LIN {X 0,Y 390.142,Z 309.368,A -85,B 0,C 180,E1 -11537.308,E2 -11537.308} C_VEL
LIN {X 0,Y 390.081,Z 309.382,A -85,B 0,C 180,E1 -11540.471,E2 -11540.471} C_VEL
LIN {X 0,Y 390.069,Z 309.39,A -85,B 0,C 180,E1 -11544.482,E2 -11544.482} C_VEL
LIN {X 0,Y 390.112,Z 309.375,A -85,B 0,C 180,E1 -11547.931,E2 -11547.931} C_VEL
LIN {X 0,Y 390.017,Z 309.4,A -85,B 0,C 180,E1 -11551.506,E2 -11551.506} C_VEL
LIN {X 0,Y 390.065,Z 309.388,A -85,B 0,C 180,E1 -11555.21,E2 -11555.21} C_VEL
LIN {X 0,Y 390.082,Z 309.386,A -85,B 0,C 180,E1 -11559.094,E2 -11559.094} C_VEL
LIN {X 0,Y 390.039,Z 309.401,A -85,B 0,C 180,E1 -11562.375,E2 -11562.375} C_VEL
LIN {X 0,Y 390.041,Z 309.396,A -85,B 0,C 180,E1 -11565.355,E2 -11565.355} C_VEL
LIN {X 0,Y 390.021,Z 309.39,A -85,B 0,C 180,E1 -11568.187,E2 -11568.187} C_VEL
LIN {X 0,Y 390.061,Z 309.392,A -85,B 0,C 180,E1 -11570.905,E2 -11570.905} C_VEL
LIN {X 0,Y 390.084,Z 309.385,A -85,B 0,C 180,E1 -11574.794,E2 -11574.794} C_VEL
LIN {X 0,Y 390.028,Z 309.401,A -85,B 0,C 180,E1 -11578.497,E2 -11578.497} C_VEL
LIN {X 0,Y 390.13,Z 309.588,A -85,B 0,C 180,E1 -11579.709,E2 -11579.709} C_VEL
LIN {X 0,Y 392.282,Z 320.516,A -85,B 0,C 180,E1 -11583.105,E2 -11583.105} C_VEL
LIN {X 0,Y 392.85,Z 325.729,A -85,B 0,C 180,E1 -11584.574,E2 -11584.574} C_VEL
LIN {X 0,Y 391.795,Z 337.996,A -85,B 0,C 180,E1 -11587.871,E2 -11587.871} C_VEL
LIN {X 0,Y 391.304,Z 343.848,A -85,B 0,C 180,E1 -11589.465,E2 -11589.465} C_VEL
LIN {X 0,Y 391.869,Z 347.073,A -85,B 0,C 180,E1 -11589.616,E2 -11589.616} C_VEL
LIN {X 0,Y 396.698,Z 373.255,A -85,B 0,C 180,E1 -11590.366,E2 -11590.366} C_VEL
LIN {X 0,Y 396.546,Z 399.29,A -85,B 0,C 180,E1 -11590.847,E2 -11590.847} C_VEL
LIN {X 0,Y 395.821,Z 450.139,A -85,B 0,C 180,E1 -11591.797,E2 -11591.797} C_VEL
LIN {X 0,Y 395.391,Z 460.446,A -85,B 0,C 180,E1 -11592.112,E2 -11592.112} C_VEL
LIN {X 0,Y 394.883,Z 469.958,A -85,B 0,C 180,E1 -11592.523,E2 -11592.523} C_VEL
LIN {X 0,Y 394.257,Z 480.039,A -85,B 0,C 180,E1 -11593.095,E2 -11593.095} C_VEL
LIN {X 0,Y 393.494,Z 489.796,A -85,B 0,C 180,E1 -11593.796,E2 -11593.796} C_VEL
LIN {X 0,Y 392.668,Z 499.864,A -85,B 0,C 180,E1 -11594.693,E2 -11594.693} C_VEL
LIN {X 0,Y 391.74,Z 510.864,A -85,B 0,C 180,E1 -11595.915,E2 -11595.915} C_VEL
LIN {X 0,Y 390.927,Z 520.506,A -85,B 0,C 180,E1 -11597.278,E2 -11597.278} C_VEL
LIN {X 0,Y 390.31,Z 526.707,A -85,B 0,C 180,E1 -11598.313,E2 -11598.313} C_VEL
LIN {X 0,Y 389.792,Z 533.245,A -85,B 0,C 180,E1 -11599.613,E2 -11599.613} C_VEL
LIN {X 0,Y 389.389,Z 537.746,A -85,B 0,C 180,E1 -11600.652,E2 -11600.652} C_VEL
LIN {X 0,Y 389.034,Z 543.238,A -85,B 0,C 180,E1 -11602.213,E2 -11602.213} C_VEL
LIN {X 0,Y 388.796,Z 547.562,A -85,B 0,C 180,E1 -11603.774,E2 -11603.774} C_VEL
LIN {X 0,Y 388.741,Z 549.929,A -85,B 0,C 180,E1 -11604.814,E2 -11604.814} C_VEL
LIN {X 0,Y 388.701,Z 551.728,A -85,B 0,C 180,E1 -11605.853,E2 -11605.853} C_VEL
LIN {X 0,Y 388.661,Z 554.171,A -85,B 0,C 180,E1 -11607.927,E2 -11607.927} C_VEL
LIN {X 0,Y 388.704,Z 554.761,A -85,B 0,C 180,E1 -11608.964,E2 -11608.964} C_VEL
LIN {X 0,Y 388.704,Z 554.761,A -85,B 0,C 180,E1 -11611.036,E2 -11611.036} C_VEL
LIN {X 0,Y 388.661,Z 554.171,A -85,B 0,C 180,E1 -11612.073,E2 -11612.073} C_VEL
LIN {X 0,Y 388.701,Z 551.728,A -85,B 0,C 180,E1 -11614.147,E2 -11614.147} C_VEL
LIN {X 0,Y 388.727,Z 548.672,A -85,B 0,C 180,E1 -11615.752,E2 -11615.752} C_VEL
LIN {X 0,Y 388.94,Z 544.792,A -85,B 0,C 180,E1 -11617.266,E2 -11617.266} C_VEL
LIN {X 0,Y 389.257,Z 539.662,A -85,B 0,C 180,E1 -11618.828,E2 -11618.828} C_VEL
LIN {X 0,Y 389.666,Z 534.4,A -85,B 0,C 180,E1 -11620.128,E2 -11620.128} C_VEL
LIN {X 0,Y 390.165,Z 528.082,A -85,B 0,C 180,E1 -11621.428,E2 -11621.428} C_VEL
LIN {X 0,Y 390.767,Z 522.133,A -85,B 0,C 180,E1 -11622.463,E2 -11622.463} C_VEL
LIN {X 0,Y 391.353,Z 515.204,A -85,B 0,C 180,E1 -11623.5,E2 -11623.5} C_VEL
LIN {X 0,Y 392.026,Z 507.023,A -85,B 0,C 180,E1 -11624.535,E2 -11624.535} C_VEL
LIN {X 0,Y 392.753,Z 498.511,A -85,B 0,C 180,E1 -11625.436,E2 -11625.436} C_VEL
LIN {X 0,Y 393.496,Z 489.796,A -85,B 0,C 180,E1 -11626.204,E2 -11626.204} C_VEL
LIN {X 0,Y 394.264,Z 480.04,A -85,B 0,C 180,E1 -11626.904,E2 -11626.904} C_VEL
LIN {X 0,Y 394.855,Z 469.958,A -85,B 0,C 180,E1 -11627.479,E2 -11627.479} C_VEL
LIN {X 0,Y 395.422,Z 460.447,A -85,B 0,C 180,E1 -11627.887,E2 -11627.887} C_VEL
LIN {X 0,Y 395.803,Z 450.139,A -85,B 0,C 180,E1 -11628.203,E2 -11628.203} C_VEL
LIN {X 0,Y 396.422,Z 404.772,A -85,B 0,C 180,E1 -11629.056,E2 -11629.056} C_VEL
LIN {X 0,Y 396.829,Z 373.982,A -85,B 0,C 180,E1 -11629.614,E2 -11629.614} C_VEL
LIN {X 0,Y 391.498,Z 345.223,A -85,B 0,C 180,E1 -11630.439,E2 -11630.439} C_VEL
LIN {X 0,Y 391.324,Z 343.641,A -85,B 0,C 180,E1 -11630.568,E2 -11630.568} C_VEL
LIN {X 0,Y 392.44,Z 331.107,A -85,B 0,C 180,E1 -11634.029,E2 -11634.029} C_VEL
LIN {X 0,Y 392.897,Z 325.998,A -85,B 0,C 180,E1 -11635.423,E2 -11635.423} C_VEL
LIN {X 0,Y 392.326,Z 320.813,A -85,B 0,C 180,E1 -11636.892,E2 -11636.892} C_VEL
LIN {X 0,Y 390.56,Z 311.768,A -85,B 0,C 180,E1 -11639.599,E2 -11639.599} C_VEL
LIN {X 0,Y 390.097,Z 309.445,A -85,B 0,C 180,E1 -11640.369,E2 -11640.369} C_VEL
LIN {X 0,Y 390.068,Z 309.4,A -85,B 0,C 180,E1 -11644.024,E2 -11644.024} C_VEL
LIN {X 0,Y 390.039,Z 309.399,A -85,B 0,C 180,E1 -11647.549,E2 -11647.549} C_VEL
LIN {X 0,Y 390.02,Z 309.382,A -85,B 0,C 180,E1 -11650.814,E2 -11650.814} C_VEL
LIN {X 0,Y 390.051,Z 309.401,A -85,B 0,C 180,E1 -11653.885,E2 -11653.885} C_VEL
LIN {X 0,Y 390.054,Z 309.395,A -85,B 0,C 180,E1 -11656.789,E2 -11656.789} C_VEL
LIN {X 0,Y 390.053,Z 309.392,A -85,B 0,C 180,E1 -11659.559,E2 -11659.559} C_VEL
LIN {X 0,Y 390.038,Z 309.398,A -85,B 0,C 180,E1 -11662.449,E2 -11662.449} C_VEL
LIN {X 0,Y 390.056,Z 309.384,A -85,B 0,C 180,E1 -11666.043,E2 -11666.043} C_VEL
LIN {X 0,Y 390.041,Z 309.399,A -85,B 0,C 180,E1 -11669.868,E2 -11669.868} C_VEL
LIN {X 0,Y 390.107,Z 309.372,A -85,B 0,C 180,E1 -11673.231,E2 -11673.231} C_VEL
LIN {X 0,Y 390.061,Z 309.393,A -85,B 0,C 180,E1 -11676.763,E2 -11676.763} C_VEL
LIN {X 0,Y 390.097,Z 309.375,A -85,B 0,C 180,E1 -11679.982,E2 -11679.982} C_VEL
LIN {X 0,Y 390.131,Z 309.374,A -85,B 0,C 180,E1 -11683.247,E2 -11683.247} C_VEL
LIN {X 0,Y 390.187,Z 309.377,A -85,B 0,C 180,E1 -11686.561,E2 -11686.561} C_VEL
LIN {X 0,Y 390.197,Z 309.351,A -85,B 0,C 180,E1 -11690.67,E2 -11690.67} C_VEL
LIN {X 0,Y 390.318,Z 309.363,A -85,B 0,C 180,E1 -11693.797,E2 -11693.797} C_VEL
LIN {X 0,Y 390.412,Z 309.342,A -85,B 0,C 180,E1 -11697.936,E2 -11697.936} C_VEL
LIN {X 0,Y 390.54,Z 309.307,A -85,B 0,C 180,E1 -11699.999,E2 -11699.999} C_VEL
LIN {X 0,Y 390.302,Z 309.359,A -85,B 0,C 180,E1 -11703.096,E2 -11703.096} C_VEL
LIN {X 0,Y 390.292,Z 309.361,A -85,B 0,C 180,E1 -11706.66,E2 -11706.66} C_VEL
LIN {X 0,Y 390.196,Z 309.354,A -85,B 0,C 180,E1 -11709.328,E2 -11709.328} C_VEL
LIN {X 0,Y 390.185,Z 309.381,A -85,B 0,C 180,E1 -11713.438,E2 -11713.438} C_VEL
LIN {X 0,Y 390.139,Z 309.375,A -85,B 0,C 180,E1 -11717.307,E2 -11717.307} C_VEL
LIN {X 0,Y 390.079,Z 309.378,A -85,B 0,C 180,E1 -11720.47,E2 -11720.47} C_VEL
LIN {X 0,Y 390.08,Z 309.394,A -85,B 0,C 180,E1 -11723.351,E2 -11723.351} C_VEL
LIN {X 0,Y 390.104,Z 309.376,A -85,B 0,C 180,E1 -11726.768,E2 -11726.768} C_VEL
LIN {X 0,Y 390.035,Z 309.398,A -85,B 0,C 180,E1 -11730.299,E2 -11730.299} C_VEL
LIN {X 0,Y 390.059,Z 309.386,A -85,B 0,C 180,E1 -11734.025,E2 -11734.025} C_VEL
LIN {X 0,Y 390.039,Z 309.399,A -85,B 0,C 180,E1 -11737.552,E2 -11737.552} C_VEL
LIN {X 0,Y 390.074,Z 309.386,A -85,B 0,C 180,E1 -11740.826,E2 -11740.826} C_VEL
LIN {X 0,Y 390.094,Z 309.391,A -85,B 0,C 180,E1 -11743.894,E2 -11743.894} C_VEL
LIN {X 0,Y 390.049,Z 309.362,A -85,B 0,C 180,E1 -11747.624,E2 -11747.624} C_VEL
LIN {X 0,Y 390.087,Z 309.392,A -85,B 0,C 180,E1 -11750.908,E2 -11750.908} C_VEL
LIN {X 0,Y 390.079,Z 309.371,A -85,B 0,C 180,E1 -11754.793,E2 -11754.793} C_VEL
LIN {X 0,Y 390.018,Z 309.404,A -85,B 0,C 180,E1 -11758.496,E2 -11758.496} C_VEL
LIN {X 0,Y 390.112,Z 309.386,A -85,B 0,C 180,E1 -11762.07,E2 -11762.07} C_VEL
LIN {X 0,Y 390.075,Z 309.396,A -85,B 0,C 180,E1 -11765.52,E2 -11765.52} C_VEL
LIN {X 0,Y 390.051,Z 309.4,A -85,B 0,C 180,E1 -11768.878,E2 -11768.878} C_VEL
LIN {X 0,Y 390.123,Z 309.392,A -85,B 0,C 180,E1 -11772.167,E2 -11772.167} C_VEL
LIN {X 0,Y 390.14,Z 309.39,A -85,B 0,C 180,E1 -11775.393,E2 -11775.393} C_VEL
LIN {X 0,Y 390.144,Z 309.389,A -85,B 0,C 180,E1 -11778.571,E2 -11778.571} C_VEL
LIN {X 0,Y 390.382,Z 309.658,A -85,B 0,C 180,E1 -11781.83,E2 -11781.83} C_VEL
LIN {X 0,Y 390.711,Z 310.916,A -85,B 0,C 180,E1 -11782.459,E2 -11782.459} C_VEL
LIN {X 0,Y 392.084,Z 313.241,A -85,B 0,C 180,E1 -11783.568,E2 -11783.568} C_VEL
LIN {X 0,Y 394.112,Z 314.918,A -85,B 0,C 180,E1 -11785.397,E2 -11785.397} C_VEL
LIN {X 0,Y 395.582,Z 315.492,A -85,B 0,C 180,E1 -11787.454,E2 -11787.454} C_VEL
LIN {X 0,Y 396.128,Z 315.931,A -85,B 0,C 180,E1 -11788.983,E2 -11788.983} C_VEL
LIN {X 0,Y 396.323,Z 315.849,A -85,B 0,C 180,E1 -11790,E2 -11790} C_VEL
LIN {X 0,Y 396.07,Z 315.804,A -85,B 0,C 180,E1 -11791.525,E2 -11791.525} C_VEL
LIN {X 0,Y 395.354,Z 315.371,A -85,B 0,C 180,E1 -11793.057,E2 -11793.057} C_VEL
LIN {X 0,Y 393.694,Z 314.658,A -85,B 0,C 180,E1 -11794.992,E2 -11794.992} C_VEL
LIN {X 0,Y 391.898,Z 313.021,A -85,B 0,C 180,E1 -11796.565,E2 -11796.565} C_VEL
LIN {X 0,Y 390.579,Z 310.503,A -85,B 0,C 180,E1 -11797.684,E2 -11797.684} C_VEL
LIN {X 0,Y 390.341,Z 309.593,A -85,B 0,C 180,E1 -11798.281,E2 -11798.281} C_VEL
LIN {X 0,Y 390.144,Z 309.389,A -85,B 0,C 180,E1 -11801.429,E2 -11801.429} C_VEL
LIN {X 0,Y 390.14,Z 309.39,A -85,B 0,C 180,E1 -11804.607,E2 -11804.607} C_VEL
LIN {X 0,Y 390.123,Z 309.392,A -85,B 0,C 180,E1 -11807.833,E2 -11807.833} C_VEL
LIN {X 0,Y 390.051,Z 309.4,A -85,B 0,C 180,E1 -11811.122,E2 -11811.122} C_VEL
LIN {X 0,Y 390.075,Z 309.396,A -85,B 0,C 180,E1 -11814.48,E2 -11814.48} C_VEL
LIN {X 0,Y 390.112,Z 309.386,A -85,B 0,C 180,E1 -11817.93,E2 -11817.93} C_VEL
LIN {X 0,Y 390.005,Z 309.398,A -85,B 0,C 180,E1 -11820.819,E2 -11820.819} C_VEL
LIN {X 0,Y 389.333,Z 309.491,A -85,B 0,C 180,E1 -11821.681,E2 -11821.681} C_VEL
LIN {X 0,Y 386.485,Z 309.833,A -85,B 0,C 180,E1 -11823.083,E2 -11823.083} C_VEL
LIN {X 0,Y 384.086,Z 310.119,A -85,B 0,C 180,E1 -11824.216,E2 -11824.216} C_VEL
LIN {X 0,Y 383.069,Z 310.243,A -85,B 0,C 180,E1 -11825.091,E2 -11825.091} C_VEL
LIN {X 0,Y 382.992,Z 310.255,A -85,B 0,C 180,E1 -11825.388,E2 -11825.388} C_VEL
LIN {X 0,Y 383,Z 310.276,A -85,B 0,C 180,E1 -11828.6,E2 -11828.6} C_VEL
LIN {X 0,Y 382.996,Z 310.242,A -85,B 0,C 180,E1 -11831.345,E2 -11831.345} C_VEL
LIN {X 0,Y 383.002,Z 310.265,A -85,B 0,C 180,E1 -11834.305,E2 -11834.305} C_VEL
LIN {X 0,Y 383.067,Z 310.27,A -85,B 0,C 180,E1 -11837.249,E2 -11837.249} C_VEL
LIN {X 0,Y 383.014,Z 310.268,A -85,B 0,C 180,E1 -11840.412,E2 -11840.412} C_VEL
LIN {X 0,Y 383.018,Z 310.267,A -85,B 0,C 180,E1 -11844.045,E2 -11844.045} C_VEL
LIN {X 0,Y 382.998,Z 310.278,A -85,B 0,C 180,E1 -11847.573,E2 -11847.573} C_VEL
LIN {X 0,Y 383.041,Z 310.256,A -85,B 0,C 180,E1 -11851.508,E2 -11851.508} C_VEL
LIN {X 0,Y 383.043,Z 310.267,A -85,B 0,C 180,E1 -11855.04,E2 -11855.04} C_VEL
LIN {X 0,Y 382.99,Z 310.274,A -85,B 0,C 180,E1 -11858.47,E2 -11858.47} C_VEL
LIN {X 0,Y 383.08,Z 310.251,A -85,B 0,C 180,E1 -11861.828,E2 -11861.828} C_VEL
LIN {X 0,Y 383.103,Z 310.266,A -85,B 0,C 180,E1 -11865.119,E2 -11865.119} C_VEL
LIN {X 0,Y 383.089,Z 310.253,A -85,B 0,C 180,E1 -11868.358,E2 -11868.358} C_VEL
LIN {X 0,Y 383.255,Z 310.232,A -85,B 0,C 180,E1 -11871.976,E2 -11871.976} C_VEL
LIN {X 0,Y 383.189,Z 310.255,A -85,B 0,C 180,E1 -11874.739,E2 -11874.739} C_VEL
LIN {X 0,Y 383.376,Z 310.216,A -85,B 0,C 180,E1 -11877.899,E2 -11877.899} C_VEL
LIN {X 0,Y 383.51,Z 310.182,A -85,B 0,C 180,E1 -11880.001,E2 -11880.001} C_VEL
LIN {X 0,Y 383.243,Z 310.245,A -85,B 0,C 180,E1 -11883.154,E2 -11883.154} C_VEL
LIN {X 0,Y 383.274,Z 310.241,A -85,B 0,C 180,E1 -11886.317,E2 -11886.317} C_VEL
LIN {X 0,Y 383.144,Z 310.228,A -85,B 0,C 180,E1 -11889.503,E2 -11889.503} C_VEL
LIN {X 0,Y 383.118,Z 310.257,A -85,B 0,C 180,E1 -11893.537,E2 -11893.537} C_VEL
LIN {X 0,Y 383.088,Z 310.246,A -85,B 0,C 180,E1 -11897.455,E2 -11897.455} C_VEL
LIN {X 0,Y 383.022,Z 310.264,A -85,B 0,C 180,E1 -11900.648,E2 -11900.648} C_VEL
LIN {X 0,Y 383.015,Z 310.271,A -85,B 0,C 180,E1 -11903.809,E2 -11903.809} C_VEL
LIN {X 0,Y 383.074,Z 310.251,A -85,B 0,C 180,E1 -11906.124,E2 -11906.124} C_VEL
LIN {X 0,Y 382.986,Z 310.275,A -85,B 0,C 180,E1 -11909.701,E2 -11909.701} C_VEL
LIN {X 0,Y 382.994,Z 310.264,A -85,B 0,C 180,E1 -11913.402,E2 -11913.402} C_VEL
LIN {X 0,Y 383.019,Z 310.271,A -85,B 0,C 180,E1 -11916.164,E2 -11916.164} C_VEL
LIN {X 0,Y 383.004,Z 310.267,A -85,B 0,C 180,E1 -11919.96,E2 -11919.96} C_VEL
LIN {X 0,Y 383.003,Z 310.274,A -85,B 0,C 180,E1 -11922.78,E2 -11922.78} C_VEL
LIN {X 0,Y 382.994,Z 310.277,A -85,B 0,C 180,E1 -11925.79,E2 -11925.79} C_VEL
LIN {X 0,Y 382.963,Z 310.263,A -85,B 0,C 180,E1 -11928.801,E2 -11928.801} C_VEL
LIN {X 0,Y 382.993,Z 310.281,A -85,B 0,C 180,E1 -11932.098,E2 -11932.098} C_VEL
LIN {X 0,Y 383.017,Z 310.272,A -85,B 0,C 180,E1 -11935.333,E2 -11935.333} C_VEL
LIN {X 0,Y 383.044,Z 310.305,A -85,B 0,C 180,E1 -11939.309,E2 -11939.309} C_VEL
LIN {X 0,Y 385.021,Z 320.33,A -85,B 0,C 180,E1 -11942.555,E2 -11942.555} C_VEL
LIN {X 0,Y 385.884,Z 326.592,A -85,B 0,C 180,E1 -11944.371,E2 -11944.371} C_VEL
LIN {X 0,Y 384.899,Z 337.805,A -85,B 0,C 180,E1 -11947.453,E2 -11947.453} C_VEL
LIN {X 0,Y 384.384,Z 343.648,A -85,B 0,C 180,E1 -11949.077,E2 -11949.077} C_VEL
LIN {X 0,Y 384.951,Z 346.904,A -85,B 0,C 180,E1 -11949.234,E2 -11949.234} C_VEL
LIN {X 0,Y 390.121,Z 374.83,A -85,B 0,C 180,E1 -11950.054,E2 -11950.054} C_VEL
LIN {X 0,Y 389.148,Z 448.615,A -85,B 0,C 180,E1 -11951.44,E2 -11951.44} C_VEL
LIN {X 0,Y 388.761,Z 458.505,A -85,B 0,C 180,E1 -11951.728,E2 -11951.728} C_VEL
LIN {X 0,Y 388.188,Z 468.477,A -85,B 0,C 180,E1 -11952.143,E2 -11952.143} C_VEL
LIN {X 0,Y 387.549,Z 478.839,A -85,B 0,C 180,E1 -11952.726,E2 -11952.726} C_VEL
LIN {X 0,Y 386.81,Z 487.97,A -85,B 0,C 180,E1 -11953.372,E2 -11953.372} C_VEL
LIN {X 0,Y 386.019,Z 496.965,A -85,B 0,C 180,E1 -11954.152,E2 -11954.152} C_VEL
LIN {X 0,Y 385.271,Z 505.694,A -85,B 0,C 180,E1 -11955.069,E2 -11955.069} C_VEL
LIN {X 0,Y 384.547,Z 513.62,A -85,B 0,C 180,E1 -11956.061,E2 -11956.061} C_VEL
LIN {X 0,Y 383.812,Z 521.938,A -85,B 0,C 180,E1 -11957.307,E2 -11957.307} C_VEL
LIN {X 0,Y 383.181,Z 527.888,A -85,B 0,C 180,E1 -11958.361,E2 -11958.361} C_VEL
LIN {X 0,Y 382.662,Z 534.206,A -85,B 0,C 180,E1 -11959.685,E2 -11959.685} C_VEL
LIN {X 0,Y 382.213,Z 539.468,A -85,B 0,C 180,E1 -11961.008,E2 -11961.008} C_VEL
LIN {X 0,Y 381.868,Z 544.597,A -85,B 0,C 180,E1 -11962.598,E2 -11962.598} C_VEL
LIN {X 0,Y 381.688,Z 547.884,A -85,B 0,C 180,E1 -11963.882,E2 -11963.882} C_VEL
LIN {X 0,Y 381.642,Z 549.735,A -85,B 0,C 180,E1 -11964.717,E2 -11964.717} C_VEL
LIN {X 0,Y 381.626,Z 551.534,A -85,B 0,C 180,E1 -11965.776,E2 -11965.776} C_VEL
LIN {X 0,Y 381.56,Z 553.977,A -85,B 0,C 180,E1 -11967.889,E2 -11967.889} C_VEL
LIN {X 0,Y 381.603,Z 554.567,A -85,B 0,C 180,E1 -11968.945,E2 -11968.945} C_VEL
LIN {X 0,Y 381.603,Z 554.567,A -85,B 0,C 180,E1 -11971.055,E2 -11971.055} C_VEL
LIN {X 0,Y 381.56,Z 553.977,A -85,B 0,C 180,E1 -11972.111,E2 -11972.111} C_VEL
LIN {X 0,Y 381.626,Z 551.534,A -85,B 0,C 180,E1 -11974.224,E2 -11974.224} C_VEL
LIN {X 0,Y 381.642,Z 549.735,A -85,B 0,C 180,E1 -11975.283,E2 -11975.283} C_VEL
LIN {X 0,Y 381.782,Z 546.127,A -85,B 0,C 180,E1 -11976.872,E2 -11976.872} C_VEL
LIN {X 0,Y 382.094,Z 541.384,A -85,B 0,C 180,E1 -11978.461,E2 -11978.461} C_VEL
LIN {X 0,Y 382.536,Z 535.361,A -85,B 0,C 180,E1 -11980.051,E2 -11980.051} C_VEL
LIN {X 0,Y 383.062,Z 529.264,A -85,B 0,C 180,E1 -11981.375,E2 -11981.375} C_VEL
LIN {X 0,Y 383.645,Z 523.565,A -85,B 0,C 180,E1 -11982.43,E2 -11982.43} C_VEL
LIN {X 0,Y 384.406,Z 515.009,A -85,B 0,C 180,E1 -11983.749,E2 -11983.749} C_VEL
LIN {X 0,Y 385.145,Z 506.829,A -85,B 0,C 180,E1 -11984.801,E2 -11984.801} C_VEL
LIN {X 0,Y 385.905,Z 498.317,A -85,B 0,C 180,E1 -11985.717,E2 -11985.717} C_VEL
LIN {X 0,Y 386.661,Z 489.602,A -85,B 0,C 180,E1 -11986.499,E2 -11986.499} C_VEL
LIN {X 0,Y 387.479,Z 479.846,A -85,B 0,C 180,E1 -11987.209,E2 -11987.209} C_VEL
LIN {X 0,Y 388.003,Z 471.051,A -85,B 0,C 180,E1 -11987.729,E2 -11987.729} C_VEL
LIN {X 0,Y 388.641,Z 461.128,A -85,B 0,C 180,E1 -11988.176,E2 -11988.176} C_VEL
LIN {X 0,Y 389.032,Z 451.277,A -85,B 0,C 180,E1 -11988.498,E2 -11988.498} C_VEL
LIN {X 0,Y 389.434,Z 428.46,A -85,B 0,C 180,E1 -11988.955,E2 -11988.955} C_VEL
LIN {X 0,Y 390.125,Z 374.714,A -85,B 0,C 180,E1 -11989.948,E2 -11989.948} C_VEL
LIN {X 0,Y 384.701,Z 345.567,A -85,B 0,C 180,E1 -11990.806,E2 -11990.806} C_VEL
LIN {X 0,Y 384.382,Z 343.646,A -85,B 0,C 180,E1 -11990.923,E2 -11990.923} C_VEL
LIN {X 0,Y 385.503,Z 331.651,A -85,B 0,C 180,E1 -11994.28,E2 -11994.28} C_VEL
LIN {X 0,Y 385.895,Z 325.829,A -85,B 0,C 180,E1 -11995.918,E2 -11995.918} C_VEL
LIN {X 0,Y 384.517,Z 317.514,A -85,B 0,C 180,E1 -11998.373,E2 -11998.373} C_VEL
LIN {X 0,Y 383.047,Z 310.296,A -85,B 0,C 180,E1 -12000.691,E2 -12000.691} C_VEL
LIN {X 0,Y 383.017,Z 310.272,A -85,B 0,C 180,E1 -12004.667,E2 -12004.667} C_VEL
LIN {X 0,Y 382.993,Z 310.281,A -85,B 0,C 180,E1 -12007.902,E2 -12007.902} C_VEL
LIN {X 0,Y 382.963,Z 310.264,A -85,B 0,C 180,E1 -12011.349,E2 -12011.349} C_VEL
LIN {X 0,Y 382.993,Z 310.276,A -85,B 0,C 180,E1 -12014.302,E2 -12014.302} C_VEL
LIN {X 0,Y 383.008,Z 310.274,A -85,B 0,C 180,E1 -12017.239,E2 -12017.239} C_VEL
LIN {X 0,Y 383.01,Z 310.267,A -85,B 0,C 180,E1 -12020.413,E2 -12020.413} C_VEL
LIN {X 0,Y 383.01,Z 310.27,A -85,B 0,C 180,E1 -12024.042,E2 -12024.042} C_VEL
LIN {X 0,Y 382.98,Z 310.272,A -85,B 0,C 180,E1 -12027.577,E2 -12027.577} C_VEL
LIN {X 0,Y 382.986,Z 310.275,A -85,B 0,C 180,E1 -12030.299,E2 -12030.299} C_VEL
LIN {X 0,Y 383.074,Z 310.252,A -85,B 0,C 180,E1 -12034.02,E2 -12034.02} C_VEL
LIN {X 0,Y 382.985,Z 310.279,A -85,B 0,C 180,E1 -12037.333,E2 -12037.333} C_VEL
LIN {X 0,Y 383.053,Z 310.25,A -85,B 0,C 180,E1 -12040.715,E2 -12040.715} C_VEL
LIN {X 0,Y 383.074,Z 310.262,A -85,B 0,C 180,E1 -12044.026,E2 -12044.026} C_VEL
LIN {X 0,Y 383.129,Z 310.257,A -85,B 0,C 180,E1 -12047.283,E2 -12047.283} C_VEL
LIN {X 0,Y 383.144,Z 310.228,A -85,B 0,C 180,E1 -12050.497,E2 -12050.497} C_VEL
LIN {X 0,Y 383.274,Z 310.241,A -85,B 0,C 180,E1 -12053.683,E2 -12053.683} C_VEL
LIN {X 0,Y 383.379,Z 310.218,A -85,B 0,C 180,E1 -12057.898,E2 -12057.898} C_VEL
LIN {X 0,Y 383.51,Z 310.182,A -85,B 0,C 180,E1 -12059.999,E2 -12059.999} C_VEL
LIN {X 0,Y 383.239,Z 310.24,A -85,B 0,C 180,E1 -12063.153,E2 -12063.153} C_VEL
LIN {X 0,Y 383.251,Z 310.238,A -85,B 0,C 180,E1 -12066.653,E2 -12066.653} C_VEL
LIN {X 0,Y 383.142,Z 310.231,A -85,B 0,C 180,E1 -12069.502,E2 -12069.502} C_VEL
LIN {X 0,Y 383.116,Z 310.261,A -85,B 0,C 180,E1 -12073.536,E2 -12073.536} C_VEL
LIN {X 0,Y 383.085,Z 310.252,A -85,B 0,C 180,E1 -12077.454,E2 -12077.454} C_VEL
LIN {X 0,Y 383.022,Z 310.258,A -85,B 0,C 180,E1 -12080.648,E2 -12080.648} C_VEL
LIN {X 0,Y 383.024,Z 310.271,A -85,B 0,C 180,E1 -12083.807,E2 -12083.807} C_VEL
LIN {X 0,Y 383.048,Z 310.251,A -85,B 0,C 180,E1 -12087.302,E2 -12087.302} C_VEL
LIN {X 0,Y 382.978,Z 310.283,A -85,B 0,C 180,E1 -12090.918,E2 -12090.918} C_VEL
LIN {X 0,Y 383.009,Z 310.262,A -85,B 0,C 180,E1 -12094.34,E2 -12094.34} C_VEL
LIN {X 0,Y 382.99,Z 310.278,A -85,B 0,C 180,E1 -12097.268,E2 -12097.268} C_VEL
LIN {X 0,Y 383.012,Z 310.268,A -85,B 0,C 180,E1 -12099.957,E2 -12099.957} C_VEL
LIN {X 0,Y 383.058,Z 310.271,A -85,B 0,C 180,E1 -12102.788,E2 -12102.788} C_VEL
LIN {X 0,Y 383.002,Z 310.264,A -85,B 0,C 180,E1 -12105.791,E2 -12105.791} C_VEL
LIN {X 0,Y 383,Z 310.243,A -85,B 0,C 180,E1 -12108.793,E2 -12108.793} C_VEL
LIN {X 0,Y 382.996,Z 310.279,A -85,B 0,C 180,E1 -12112.096,E2 -12112.096} C_VEL
LIN {X 0,Y 383.012,Z 310.249,A -85,B 0,C 180,E1 -12115.332,E2 -12115.332} C_VEL
LIN {X 0,Y 382.977,Z 310.276,A -85,B 0,C 180,E1 -12119.082,E2 -12119.082} C_VEL
LIN {X 0,Y 383.051,Z 310.273,A -85,B 0,C 180,E1 -12122.698,E2 -12122.698} C_VEL
LIN {X 0,Y 383.047,Z 310.272,A -85,B 0,C 180,E1 -12125.04,E2 -12125.04} C_VEL
LIN {X 0,Y 382.988,Z 310.281,A -85,B 0,C 180,E1 -12128.469,E2 -12128.469} C_VEL
LIN {X 0,Y 383.085,Z 310.269,A -85,B 0,C 180,E1 -12131.828,E2 -12131.828} C_VEL
LIN {X 0,Y 383.106,Z 310.266,A -85,B 0,C 180,E1 -12135.118,E2 -12135.118} C_VEL
LIN {X 0,Y 383.113,Z 310.39,A -85,B 0,C 180,E1 -12138.359,E2 -12138.359} C_VEL
LIN {X 0,Y 383.304,Z 311.255,A -85,B 0,C 180,E1 -12138.867,E2 -12138.867} C_VEL
LIN {X 0,Y 384.444,Z 313.6,A -85,B 0,C 180,E1 -12139.533,E2 -12139.533} C_VEL
LIN {X 0,Y 386.583,Z 315.496,A -85,B 0,C 180,E1 -12140.583,E2 -12140.583} C_VEL
LIN {X 0,Y 388.922,Z 316.83,A -85,B 0,C 180,E1 -12141.896,E2 -12141.896} C_VEL
LIN {X 0,Y 390.34,Z 319.396,A -85,B 0,C 180,E1 -12142.955,E2 -12142.955} C_VEL
LIN {X 0,Y 391.933,Z 321.071,A -85,B 0,C 180,E1 -12144.211,E2 -12144.211} C_VEL
LIN {X 0,Y 393.229,Z 321.964,A -85,B 0,C 180,E1 -12145.387,E2 -12145.387} C_VEL
LIN {X 0,Y 394.719,Z 322.512,A -85,B 0,C 180,E1 -12147.449,E2 -12147.449} C_VEL
LIN {X 0,Y 395.266,Z 322.978,A -85,B 0,C 180,E1 -12148.981,E2 -12148.981} C_VEL
LIN {X 0,Y 395.458,Z 322.896,A -85,B 0,C 180,E1 -12150,E2 -12150} C_VEL
LIN {X 0,Y 395.202,Z 322.853,A -85,B 0,C 180,E1 -12151.529,E2 -12151.529} C_VEL
LIN {X 0,Y 394.244,Z 322.355,A -85,B 0,C 180,E1 -12153.368,E2 -12153.368} C_VEL
LIN {X 0,Y 392.65,Z 321.62,A -85,B 0,C 180,E1 -12155.134,E2 -12155.134} C_VEL
LIN {X 0,Y 390.787,Z 319.981,A -85,B 0,C 180,E1 -12156.713,E2 -12156.713} C_VEL
LIN {X 0,Y 389.247,Z 317.413,A -85,B 0,C 180,E1 -12157.901,E2 -12157.901} C_VEL
LIN {X 0,Y 388.306,Z 316.316,A -85,B 0,C 180,E1 -12158.456,E2 -12158.456} C_VEL
LIN {X 0,Y 385.837,Z 315.008,A -85,B 0,C 180,E1 -12159.766,E2 -12159.766} C_VEL
LIN {X 0,Y 383.934,Z 312.791,A -85,B 0,C 180,E1 -12160.747,E2 -12160.747} C_VEL
LIN {X 0,Y 383.222,Z 310.964,A -85,B 0,C 180,E1 -12161.236,E2 -12161.236} C_VEL
LIN {X 0,Y 383.115,Z 310.297,A -85,B 0,C 180,E1 -12161.91,E2 -12161.91} C_VEL
LIN {X 0,Y 383.106,Z 310.266,A -85,B 0,C 180,E1 -12164.882,E2 -12164.882} C_VEL
LIN {X 0,Y 383.085,Z 310.268,A -85,B 0,C 180,E1 -12168.172,E2 -12168.172} C_VEL
LIN {X 0,Y 382.988,Z 310.281,A -85,B 0,C 180,E1 -12171.531,E2 -12171.531} C_VEL
LIN {X 0,Y 383.047,Z 310.272,A -85,B 0,C 180,E1 -12174.96,E2 -12174.96} C_VEL
LIN {X 0,Y 383.024,Z 310.265,A -85,B 0,C 180,E1 -12178.27,E2 -12178.27} C_VEL
LIN {X 0,Y 383.003,Z 310.275,A -85,B 0,C 180,E1 -12182.149,E2 -12182.149} C_VEL
LIN {X 0,Y 382.992,Z 310.255,A -85,B 0,C 180,E1 -12185.388,E2 -12185.388} C_VEL
LIN {X 0,Y 382.353,Z 310.349,A -85,B 0,C 180,E1 -12186.266,E2 -12186.266} C_VEL
LIN {X 0,Y 379.546,Z 310.71,A -85,B 0,C 180,E1 -12187.694,E2 -12187.694} C_VEL
LIN {X 0,Y 377.141,Z 311.009,A -85,B 0,C 180,E1 -12188.848,E2 -12188.848} C_VEL
LIN {X 0,Y 376.083,Z 311.128,A -85,B 0,C 180,E1 -12189.74,E2 -12189.74} C_VEL
LIN {X 0,Y 375.985,Z 311.134,A -85,B 0,C 180,E1 -12190.042,E2 -12190.042} C_VEL
LIN {X 0,Y 375.93,Z 311.133,A -85,B 0,C 180,E1 -12193.765,E2 -12193.765} C_VEL
LIN {X 0,Y 375.981,Z 311.151,A -85,B 0,C 180,E1 -12196.802,E2 -12196.802} C_VEL
LIN {X 0,Y 375.991,Z 311.143,A -85,B 0,C 180,E1 -12200.027,E2 -12200.027} C_VEL
LIN {X 0,Y 375.957,Z 311.15,A -85,B 0,C 180,E1 -12203.495,E2 -12203.495} C_VEL
LIN {X 0,Y 375.951,Z 311.142,A -85,B 0,C 180,E1 -12205.889,E2 -12205.889} C_VEL
LIN {X 0,Y 375.96,Z 311.151,A -85,B 0,C 180,E1 -12209.688,E2 -12209.688} C_VEL
LIN {X 0,Y 375.993,Z 311.131,A -85,B 0,C 180,E1 -12212.142,E2 -12212.142} C_VEL
LIN {X 0,Y 375.997,Z 311.14,A -85,B 0,C 180,E1 -12214.539,E2 -12214.539} C_VEL
LIN {X 0,Y 375.959,Z 311.148,A -85,B 0,C 180,E1 -12218.046,E2 -12218.046} C_VEL
LIN {X 0,Y 376.014,Z 311.126,A -85,B 0,C 180,E1 -12221.474,E2 -12221.474} C_VEL
LIN {X 0,Y 376.05,Z 311.143,A -85,B 0,C 180,E1 -12224.833,E2 -12224.833} C_VEL
LIN {X 0,Y 376.042,Z 311.132,A -85,B 0,C 180,E1 -12228.137,E2 -12228.137} C_VEL
LIN {X 0,Y 376.21,Z 311.109,A -85,B 0,C 180,E1 -12231.919,E2 -12231.919} C_VEL
LIN {X 0,Y 376.162,Z 311.129,A -85,B 0,C 180,E1 -12234.64,E2 -12234.64} C_VEL
LIN {X 0,Y 376.343,Z 311.092,A -85,B 0,C 180,E1 -12237.86,E2 -12237.86} C_VEL
LIN {X 0,Y 376.48,Z 311.057,A -85,B 0,C 180,E1 -12240.001,E2 -12240.001} C_VEL
LIN {X 0,Y 376.181,Z 311.125,A -85,B 0,C 180,E1 -12243.214,E2 -12243.214} C_VEL
LIN {X 0,Y 376.233,Z 311.116,A -85,B 0,C 180,E1 -12246.436,E2 -12246.436} C_VEL
LIN {X 0,Y 376.112,Z 311.104,A -85,B 0,C 180,E1 -12249.682,E2 -12249.682} C_VEL
LIN {X 0,Y 376.082,Z 311.134,A -85,B 0,C 180,E1 -12253.658,E2 -12253.658} C_VEL
LIN {X 0,Y 376.036,Z 311.124,A -85,B 0,C 180,E1 -12257.608,E2 -12257.608} C_VEL
LIN {X 0,Y 375.972,Z 311.145,A -85,B 0,C 180,E1 -12260.833,E2 -12260.833} C_VEL
LIN {X 0,Y 375.981,Z 311.147,A -85,B 0,C 180,E1 -12264.283,E2 -12264.283} C_VEL
LIN {X 0,Y 376.014,Z 311.126,A -85,B 0,C 180,E1 -12266.653,E2 -12266.653} C_VEL
LIN {X 0,Y 375.959,Z 311.156,A -85,B 0,C 180,E1 -12270.314,E2 -12270.314} C_VEL
LIN {X 0,Y 375.952,Z 311.139,A -85,B 0,C 180,E1 -12274.113,E2 -12274.113} C_VEL
LIN {X 0,Y 375.945,Z 311.156,A -85,B 0,C 180,E1 -12276.743,E2 -12276.743} C_VEL
LIN {X 0,Y 375.984,Z 311.141,A -85,B 0,C 180,E1 -12279.971,E2 -12279.971} C_VEL
LIN {X 0,Y 375.927,Z 311.155,A -85,B 0,C 180,E1 -12283.767,E2 -12283.767} C_VEL
LIN {X 0,Y 375.932,Z 311.156,A -85,B 0,C 180,E1 -12286.812,E2 -12286.812} C_VEL
LIN {X 0,Y 375.936,Z 311.143,A -85,B 0,C 180,E1 -12290.535,E2 -12290.535} C_VEL
LIN {X 0,Y 375.962,Z 311.144,A -85,B 0,C 180,E1 -12293.497,E2 -12293.497} C_VEL
LIN {X 0,Y 375.96,Z 311.156,A -85,B 0,C 180,E1 -12295.89,E2 -12295.89} C_VEL
LIN {X 0,Y 376.018,Z 311.368,A -85,B 0,C 180,E1 -12299.097,E2 -12299.097} C_VEL
LIN {X 0,Y 377.992,Z 321.19,A -85,B 0,C 180,E1 -12302.302,E2 -12302.302} C_VEL
LIN {X 0,Y 378.922,Z 327.455,A -85,B 0,C 180,E1 -12304.16,E2 -12304.16} C_VEL
LIN {X 0,Y 378.047,Z 337.614,A -85,B 0,C 180,E1 -12307.021,E2 -12307.021} C_VEL
LIN {X 0,Y 377.477,Z 343.493,A -85,B 0,C 180,E1 -12308.682,E2 -12308.682} C_VEL
LIN {X 0,Y 378.326,Z 347.873,A -85,B 0,C 180,E1 -12308.876,E2 -12308.876} C_VEL
LIN {X 0,Y 383.369,Z 375.316,A -85,B 0,C 180,E1 -12309.701,E2 -12309.701} C_VEL
LIN {X 0,Y 382.755,Z 425.441,A -85,B 0,C 180,E1 -12310.646,E2 -12310.646} C_VEL
LIN {X 0,Y 382.383,Z 449.752,A -85,B 0,C 180,E1 -12311.134,E2 -12311.134} C_VEL
LIN {X 0,Y 381.934,Z 460.059,A -85,B 0,C 180,E1 -12311.459,E2 -12311.459} C_VEL
LIN {X 0,Y 381.348,Z 469.57,A -85,B 0,C 180,E1 -12311.881,E2 -12311.881} C_VEL
LIN {X 0,Y 380.777,Z 478.645,A -85,B 0,C 180,E1 -12312.409,E2 -12312.409} C_VEL
LIN {X 0,Y 379.995,Z 487.776,A -85,B 0,C 180,E1 -12313.065,E2 -12313.065} C_VEL
LIN {X 0,Y 379.198,Z 496.772,A -85,B 0,C 180,E1 -12313.859,E2 -12313.859} C_VEL
LIN {X 0,Y 378.375,Z 505.499,A -85,B 0,C 180,E1 -12314.79,E2 -12314.79} C_VEL
LIN {X 0,Y 377.615,Z 513.589,A -85,B 0,C 180,E1 -12315.823,E2 -12315.823} C_VEL
LIN {X 0,Y 376.861,Z 521.744,A -85,B 0,C 180,E1 -12317.069,E2 -12317.069} C_VEL
LIN {X 0,Y 376.213,Z 527.693,A -85,B 0,C 180,E1 -12318.142,E2 -12318.142} C_VEL
LIN {X 0,Y 375.651,Z 534.011,A -85,B 0,C 180,E1 -12319.49,E2 -12319.49} C_VEL
LIN {X 0,Y 375.168,Z 539.273,A -85,B 0,C 180,E1 -12320.838,E2 -12320.838} C_VEL
LIN {X 0,Y 374.802,Z 544.403,A -85,B 0,C 180,E1 -12322.458,E2 -12322.458} C_VEL
LIN {X 0,Y 374.583,Z 548.07,A -85,B 0,C 180,E1 -12323.935,E2 -12323.935} C_VEL
LIN {X 0,Y 374.53,Z 551.34,A -85,B 0,C 180,E1 -12325.695,E2 -12325.695} C_VEL
LIN {X 0,Y 374.459,Z 553.783,A -85,B 0,C 180,E1 -12327.849,E2 -12327.849} C_VEL
LIN {X 0,Y 374.503,Z 554.373,A -85,B 0,C 180,E1 -12328.925,E2 -12328.925} C_VEL
LIN {X 0,Y 374.503,Z 554.373,A -85,B 0,C 180,E1 -12331.075,E2 -12331.075} C_VEL
LIN {X 0,Y 374.459,Z 553.783,A -85,B 0,C 180,E1 -12332.151,E2 -12332.151} C_VEL
LIN {X 0,Y 374.53,Z 551.34,A -85,B 0,C 180,E1 -12334.305,E2 -12334.305} C_VEL
LIN {X 0,Y 374.583,Z 548.071,A -85,B 0,C 180,E1 -12336.065,E2 -12336.065} C_VEL
LIN {X 0,Y 374.802,Z 544.403,A -85,B 0,C 180,E1 -12337.542,E2 -12337.542} C_VEL
LIN {X 0,Y 375.168,Z 539.273,A -85,B 0,C 180,E1 -12339.162,E2 -12339.162} C_VEL
LIN {X 0,Y 375.651,Z 534.011,A -85,B 0,C 180,E1 -12340.51,E2 -12340.51} C_VEL
LIN {X 0,Y 376.21,Z 527.693,A -85,B 0,C 180,E1 -12341.858,E2 -12341.858} C_VEL
LIN {X 0,Y 376.886,Z 521.744,A -85,B 0,C 180,E1 -12342.93,E2 -12342.93} C_VEL
LIN {X 0,Y 377.61,Z 513.601,A -85,B 0,C 180,E1 -12344.175,E2 -12344.175} C_VEL
LIN {X 0,Y 378.499,Z 504.365,A -85,B 0,C 180,E1 -12345.342,E2 -12345.342} C_VEL
LIN {X 0,Y 379.465,Z 494.069,A -85,B 0,C 180,E1 -12346.406,E2 -12346.406} C_VEL
LIN {X 0,Y 380.5,Z 481.664,A -85,B 0,C 180,E1 -12347.397,E2 -12347.397} C_VEL
LIN {X 0,Y 381.253,Z 470.857,A -85,B 0,C 180,E1 -12348.054,E2 -12348.054} C_VEL
LIN {X 0,Y 381.903,Z 460.934,A -85,B 0,C 180,E1 -12348.508,E2 -12348.508} C_VEL
LIN {X 0,Y 382.319,Z 451.083,A -85,B 0,C 180,E1 -12348.834,E2 -12348.834} C_VEL
LIN {X 0,Y 382.736,Z 428.267,A -85,B 0,C 180,E1 -12349.3,E2 -12349.3} C_VEL
LIN {X 0,Y 383.414,Z 375.322,A -85,B 0,C 180,E1 -12350.296,E2 -12350.296} C_VEL
LIN {X 0,Y 377.919,Z 345.99,A -85,B 0,C 180,E1 -12351.185,E2 -12351.185} C_VEL
LIN {X 0,Y 377.463,Z 343.514,A -85,B 0,C 180,E1 -12351.314,E2 -12351.314} C_VEL
LIN {X 0,Y 378.688,Z 331.19,A -85,B 0,C 180,E1 -12354.827,E2 -12354.827} C_VEL
LIN {X 0,Y 378.888,Z 326.68,A -85,B 0,C 180,E1 -12356.138,E2 -12356.138} C_VEL
LIN {X 0,Y 377.297,Z 317.571,A -85,B 0,C 180,E1 -12358.897,E2 -12358.897} C_VEL
LIN {X 0,Y 375.984,Z 311.171,A -85,B 0,C 180,E1 -12361.021,E2 -12361.021} C_VEL
LIN {X 0,Y 375.979,Z 311.148,A -85,B 0,C 180,E1 -12364.666,E2 -12364.666} C_VEL
LIN {X 0,Y 375.937,Z 311.156,A -85,B 0,C 180,E1 -12368.262,E2 -12368.262} C_VEL
LIN {X 0,Y 375.918,Z 311.143,A -85,B 0,C 180,E1 -12371.597,E2 -12371.597} C_VEL
LIN {X 0,Y 375.924,Z 311.155,A -85,B 0,C 180,E1 -12374.73,E2 -12374.73} C_VEL
LIN {X 0,Y 375.931,Z 311.154,A -85,B 0,C 180,E1 -12378.398,E2 -12378.398} C_VEL
LIN {X 0,Y 375.968,Z 311.15,A -85,B 0,C 180,E1 -12381.729,E2 -12381.729} C_VEL
LIN {X 0,Y 375.97,Z 311.14,A -85,B 0,C 180,E1 -12385.333,E2 -12385.333} C_VEL
LIN {X 0,Y 375.952,Z 311.152,A -85,B 0,C 180,E1 -12388.437,E2 -12388.437} C_VEL
LIN {X 0,Y 375.977,Z 311.135,A -85,B 0,C 180,E1 -12392.139,E2 -12392.139} C_VEL
LIN {X 0,Y 375.999,Z 311.136,A -85,B 0,C 180,E1 -12394.538,E2 -12394.538} C_VEL
LIN {X 0,Y 375.95,Z 311.15,A -85,B 0,C 180,E1 -12398.044,E2 -12398.044} C_VEL
LIN {X 0,Y 376.002,Z 311.123,A -85,B 0,C 180,E1 -12401.472,E2 -12401.472} C_VEL
LIN {X 0,Y 376.051,Z 311.136,A -85,B 0,C 180,E1 -12404.832,E2 -12404.832} C_VEL
LIN {X 0,Y 376.042,Z 311.131,A -85,B 0,C 180,E1 -12408.136,E2 -12408.136} C_VEL
LIN {X 0,Y 376.211,Z 311.105,A -85,B 0,C 180,E1 -12411.918,E2 -12411.918} C_VEL
LIN {X 0,Y 376.162,Z 311.125,A -85,B 0,C 180,E1 -12414.639,E2 -12414.639} C_VEL
LIN {X 0,Y 376.345,Z 311.094,A -85,B 0,C 180,E1 -12417.859,E2 -12417.859} C_VEL
LIN {X 0,Y 376.48,Z 311.057,A -85,B 0,C 180,E1 -12419.999,E2 -12419.999} C_VEL
LIN {X 0,Y 376.177,Z 311.12,A -85,B 0,C 180,E1 -12423.212,E2 -12423.212} C_VEL
LIN {X 0,Y 376.215,Z 311.116,A -85,B 0,C 180,E1 -12426.642,E2 -12426.642} C_VEL
LIN {X 0,Y 376.11,Z 311.105,A -85,B 0,C 180,E1 -12429.681,E2 -12429.681} C_VEL
LIN {X 0,Y 376.08,Z 311.137,A -85,B 0,C 180,E1 -12433.657,E2 -12433.657} C_VEL
LIN {X 0,Y 376.035,Z 311.129,A -85,B 0,C 180,E1 -12437.607,E2 -12437.607} C_VEL
LIN {X 0,Y 375.969,Z 311.138,A -85,B 0,C 180,E1 -12440.832,E2 -12440.832} C_VEL
LIN {X 0,Y 375.985,Z 311.149,A -85,B 0,C 180,E1 -12444.281,E2 -12444.281} C_VEL
LIN {X 0,Y 376.011,Z 311.131,A -85,B 0,C 180,E1 -12446.652,E2 -12446.652} C_VEL
LIN {X 0,Y 375.968,Z 311.145,A -85,B 0,C 180,E1 -12449.079,E2 -12449.079} C_VEL
LIN {X 0,Y 375.946,Z 311.15,A -85,B 0,C 180,E1 -12452.828,E2 -12452.828} C_VEL
LIN {X 0,Y 375.95,Z 311.146,A -85,B 0,C 180,E1 -12455.415,E2 -12455.415} C_VEL
LIN {X 0,Y 375.97,Z 311.154,A -85,B 0,C 180,E1 -12458.271,E2 -12458.271} C_VEL
LIN {X 0,Y 375.981,Z 311.144,A -85,B 0,C 180,E1 -12461.61,E2 -12461.61} C_VEL
LIN {X 0,Y 375.963,Z 311.143,A -85,B 0,C 180,E1 -12465.262,E2 -12465.262} C_VEL
LIN {X 0,Y 375.968,Z 311.122,A -85,B 0,C 180,E1 -12469.138,E2 -12469.138} C_VEL
LIN {X 0,Y 375.96,Z 311.154,A -85,B 0,C 180,E1 -12471.912,E2 -12471.912} C_VEL
LIN {X 0,Y 375.973,Z 311.125,A -85,B 0,C 180,E1 -12475.333,E2 -12475.333} C_VEL
LIN {X 0,Y 375.952,Z 311.157,A -85,B 0,C 180,E1 -12478.438,E2 -12478.438} C_VEL
LIN {X 0,Y 375.977,Z 311.147,A -85,B 0,C 180,E1 -12482.141,E2 -12482.141} C_VEL
LIN {X 0,Y 376.001,Z 311.151,A -85,B 0,C 180,E1 -12484.539,E2 -12484.539} C_VEL
LIN {X 0,Y 375.958,Z 311.157,A -85,B 0,C 180,E1 -12488.046,E2 -12488.046} C_VEL
LIN {X 0,Y 376.019,Z 311.148,A -85,B 0,C 180,E1 -12491.474,E2 -12491.474} C_VEL
LIN {X 0,Y 376.054,Z 311.144,A -85,B 0,C 180,E1 -12494.833,E2 -12494.833} C_VEL
LIN {X 0,Y 376.112,Z 311.433,A -85,B 0,C 180,E1 -12496.109,E2 -12496.109} C_VEL
LIN {X 0,Y 376.404,Z 312.527,A -85,B 0,C 180,E1 -12496.467,E2 -12496.467} C_VEL
LIN {X 0,Y 377.861,Z 315.028,A -85,B 0,C 180,E1 -12497.104,E2 -12497.104} C_VEL
LIN {X 0,Y 380.043,Z 316.684,A -85,B 0,C 180,E1 -12497.946,E2 -12497.946} C_VEL
LIN {X 0,Y 381.205,Z 317.437,A -85,B 0,C 180,E1 -12498.434,E2 -12498.434} C_VEL
LIN {X 0,Y 382.765,Z 319.998,A -85,B 0,C 180,E1 -12499.152,E2 -12499.152} C_VEL
LIN {X 0,Y 384.676,Z 321.973,A -85,B 0,C 180,E1 -12500.12,E2 -12500.12} C_VEL
LIN {X 0,Y 387.592,Z 323.677,A -85,B 0,C 180,E1 -12501.659,E2 -12501.659} C_VEL
LIN {X 0,Y 389.285,Z 326.436,A -85,B 0,C 180,E1 -12502.842,E2 -12502.842} C_VEL
LIN {X 0,Y 391.04,Z 328.14,A -85,B 0,C 180,E1 -12504.198,E2 -12504.198} C_VEL
LIN {X 0,Y 392.343,Z 329.01,A -85,B 0,C 180,E1 -12505.377,E2 -12505.377} C_VEL
LIN {X 0,Y 393.615,Z 329.434,A -85,B 0,C 180,E1 -12506.93,E2 -12506.93} C_VEL
LIN {X 0,Y 394.407,Z 330.003,A -85,B 0,C 180,E1 -12508.979,E2 -12508.979} C_VEL
LIN {X 0,Y 394.593,Z 329.943,A -85,B 0,C 180,E1 -12510,E2 -12510} C_VEL
LIN {X 0,Y 394.096,Z 329.716,A -85,B 0,C 180,E1 -12512.044,E2 -12512.044} C_VEL
LIN {X 0,Y 393.066,Z 329.32,A -85,B 0,C 180,E1 -12513.725,E2 -12513.725} C_VEL
LIN {X 0,Y 391.76,Z 328.66,A -85,B 0,C 180,E1 -12515.146,E2 -12515.146} C_VEL
LIN {X 0,Y 389.867,Z 327.118,A -85,B 0,C 180,E1 -12516.729,E2 -12516.729} C_VEL
LIN {X 0,Y 388.033,Z 324.485,A -85,B 0,C 180,E1 -12518.061,E2 -12518.061} C_VEL
LIN {X 0,Y 387.369,Z 323.386,A -85,B 0,C 180,E1 -12518.477,E2 -12518.477} C_VEL
LIN {X 0,Y 384.676,Z 321.972,A -85,B 0,C 180,E1 -12519.88,E2 -12519.88} C_VEL
LIN {X 0,Y 382.448,Z 319.601,A -85,B 0,C 180,E1 -12520.991,E2 -12520.991} C_VEL
LIN {X 0,Y 380.868,Z 317.115,A -85,B 0,C 180,E1 -12521.711,E2 -12521.711} C_VEL
LIN {X 0,Y 378.467,Z 315.611,A -85,B 0,C 180,E1 -12522.671,E2 -12522.671} C_VEL
LIN {X 0,Y 376.702,Z 313.283,A -85,B 0,C 180,E1 -12523.377,E2 -12523.377} C_VEL
LIN {X 0,Y 376.2,Z 311.747,A -85,B 0,C 180,E1 -12523.729,E2 -12523.729} C_VEL
LIN {X 0,Y 376.064,Z 311.166,A -85,B 0,C 180,E1 -12524.336,E2 -12524.336} C_VEL
LIN {X 0,Y 376.039,Z 311.146,A -85,B 0,C 180,E1 -12527.607,E2 -12527.607} C_VEL
LIN {X 0,Y 375.973,Z 311.154,A -85,B 0,C 180,E1 -12530.832,E2 -12530.832} C_VEL
LIN {X 0,Y 375.989,Z 311.151,A -85,B 0,C 180,E1 -12534.281,E2 -12534.281} C_VEL
LIN {X 0,Y 376.014,Z 311.148,A -85,B 0,C 180,E1 -12536.652,E2 -12536.652} C_VEL
LIN {X 0,Y 375.958,Z 311.144,A -85,B 0,C 180,E1 -12540.312,E2 -12540.312} C_VEL
LIN {X 0,Y 375.953,Z 311.129,A -85,B 0,C 180,E1 -12544.111,E2 -12544.111} C_VEL
LIN {X 0,Y 375.948,Z 311.15,A -85,B 0,C 180,E1 -12546.741,E2 -12546.741} C_VEL
LIN {X 0,Y 375.985,Z 311.134,A -85,B 0,C 180,E1 -12550.042,E2 -12550.042} C_VEL
LIN {X 0,Y 375.269,Z 311.208,A -85,B 0,C 180,E1 -12550.936,E2 -12550.936} C_VEL
LIN {X 0,Y 372.36,Z 311.562,A -85,B 0,C 180,E1 -12552.388,E2 -12552.388} C_VEL
LIN {X 0,Y 369.954,Z 311.873,A -85,B 0,C 180,E1 -12553.562,E2 -12553.562} C_VEL
LIN {X 0,Y 368.969,Z 312.013,A -85,B 0,C 180,E1 -12554.471,E2 -12554.471} C_VEL
LIN {X 0,Y 368.913,Z 312.02,A -85,B 0,C 180,E1 -12554.778,E2 -12554.778} C_VEL
LIN {X 0,Y 368.933,Z 312.022,A -85,B 0,C 180,E1 -12558.185,E2 -12558.185} C_VEL
LIN {X 0,Y 368.905,Z 312.033,A -85,B 0,C 180,E1 -12561.359,E2 -12561.359} C_VEL
LIN {X 0,Y 368.928,Z 312.015,A -85,B 0,C 180,E1 -12565.146,E2 -12565.146} C_VEL
LIN {X 0,Y 368.921,Z 312.034,A -85,B 0,C 180,E1 -12569.046,E2 -12569.046} C_VEL
LIN {X 0,Y 368.978,Z 312.007,A -85,B 0,C 180,E1 -12571.565,E2 -12571.565} C_VEL
LIN {X 0,Y 368.949,Z 312.025,A -85,B 0,C 180,E1 -12575.225,E2 -12575.225} C_VEL
LIN {X 0,Y 368.929,Z 312.017,A -85,B 0,C 180,E1 -12578.973,E2 -12578.973} C_VEL
LIN {X 0,Y 368.982,Z 312.006,A -85,B 0,C 180,E1 -12582.257,E2 -12582.257} C_VEL
LIN {X 0,Y 369.028,Z 312.015,A -85,B 0,C 180,E1 -12586.228,E2 -12586.228} C_VEL
LIN {X 0,Y 369.059,Z 311.982,A -85,B 0,C 180,E1 -12590.132,E2 -12590.132} C_VEL
LIN {X 0,Y 369.192,Z 311.994,A -85,B 0,C 180,E1 -12593.442,E2 -12593.442} C_VEL
LIN {X 0,Y 369.308,Z 311.968,A -85,B 0,C 180,E1 -12597.819,E2 -12597.819} C_VEL
LIN {X 0,Y 369.449,Z 311.932,A -85,B 0,C 180,E1 -12600.001,E2 -12600.001} C_VEL
LIN {X 0,Y 369.31,Z 311.97,A -85,B 0,C 180,E1 -12602.182,E2 -12602.182} C_VEL
LIN {X 0,Y 369.193,Z 311.99,A -85,B 0,C 180,E1 -12606.559,E2 -12606.559} C_VEL
LIN {X 0,Y 369.06,Z 311.982,A -85,B 0,C 180,E1 -12609.869,E2 -12609.869} C_VEL
LIN {X 0,Y 369.03,Z 312.012,A -85,B 0,C 180,E1 -12613.773,E2 -12613.773} C_VEL
LIN {X 0,Y 368.995,Z 312,A -85,B 0,C 180,E1 -12617.769,E2 -12617.769} C_VEL
LIN {X 0,Y 368.903,Z 312.026,A -85,B 0,C 180,E1 -12621.222,E2 -12621.222} C_VEL
LIN {X 0,Y 368.948,Z 312.017,A -85,B 0,C 180,E1 -12624.777,E2 -12624.777} C_VEL
LIN {X 0,Y 368.957,Z 312.006,A -85,B 0,C 180,E1 -12627.205,E2 -12627.205} C_VEL
LIN {X 0,Y 368.925,Z 312.028,A -85,B 0,C 180,E1 -12630.955,E2 -12630.955} C_VEL
LIN {X 0,Y 368.919,Z 312.021,A -85,B 0,C 180,E1 -12635.001,E2 -12635.001} C_VEL
LIN {X 0,Y 368.902,Z 312.026,A -85,B 0,C 180,E1 -12638.641,E2 -12638.641} C_VEL
LIN {X 0,Y 368.878,Z 312.036,A -85,B 0,C 180,E1 -12642.01,E2 -12642.01} C_VEL
LIN {X 0,Y 368.877,Z 312.032,A -85,B 0,C 180,E1 -12645.177,E2 -12645.177} C_VEL
LIN {X 0,Y 368.869,Z 312.023,A -85,B 0,C 180,E1 -12648.177,E2 -12648.177} C_VEL
LIN {X 0,Y 368.877,Z 312.033,A -85,B 0,C 180,E1 -12651.367,E2 -12651.367} C_VEL
LIN {X 0,Y 368.936,Z 312.022,A -85,B 0,C 180,E1 -12655.147,E2 -12655.147} C_VEL
LIN {X 0,Y 368.945,Z 312.174,A -85,B 0,C 180,E1 -12658.731,E2 -12658.731} C_VEL
LIN {X 0,Y 370.715,Z 321.003,A -85,B 0,C 180,E1 -12661.71,E2 -12661.71} C_VEL
LIN {X 0,Y 371.939,Z 328.318,A -85,B 0,C 180,E1 -12663.94,E2 -12663.94} C_VEL
LIN {X 0,Y 371.38,Z 335.465,A -85,B 0,C 180,E1 -12665.992,E2 -12665.992} C_VEL
LIN {X 0,Y 370.575,Z 343.376,A -85,B 0,C 180,E1 -12668.278,E2 -12668.278} C_VEL
LIN {X 0,Y 371.888,Z 350.015,A -85,B 0,C 180,E1 -12668.54,E2 -12668.54} C_VEL
LIN {X 0,Y 376.825,Z 377.051,A -85,B 0,C 180,E1 -12669.371,E2 -12669.371} C_VEL
LIN {X 0,Y 375.683,Z 449.559,A -85,B 0,C 180,E1 -12670.784,E2 -12670.784} C_VEL
LIN {X 0,Y 375.23,Z 459.866,A -85,B 0,C 180,E1 -12671.115,E2 -12671.115} C_VEL
LIN {X 0,Y 374.594,Z 469.376,A -85,B 0,C 180,E1 -12671.543,E2 -12671.543} C_VEL
LIN {X 0,Y 373.989,Z 478.45,A -85,B 0,C 180,E1 -12672.079,E2 -12672.079} C_VEL
LIN {X 0,Y 373.193,Z 487.581,A -85,B 0,C 180,E1 -12672.747,E2 -12672.747} C_VEL
LIN {X 0,Y 372.389,Z 496.578,A -85,B 0,C 180,E1 -12673.556,E2 -12673.556} C_VEL
LIN {X 0,Y 371.499,Z 505.305,A -85,B 0,C 180,E1 -12674.502,E2 -12674.502} C_VEL
LIN {X 0,Y 370.781,Z 512.838,A -85,B 0,C 180,E1 -12675.475,E2 -12675.475} C_VEL
LIN {X 0,Y 370.105,Z 519.922,A -85,B 0,C 180,E1 -12676.549,E2 -12676.549} C_VEL
LIN {X 0,Y 369.435,Z 526.124,A -85,B 0,C 180,E1 -12677.643,E2 -12677.643} C_VEL
LIN {X 0,Y 368.701,Z 532.659,A -85,B 0,C 180,E1 -12679.012,E2 -12679.012} C_VEL
LIN {X 0,Y 368.292,Z 537.162,A -85,B 0,C 180,E1 -12680.111,E2 -12680.111} C_VEL
LIN {X 0,Y 367.857,Z 542.654,A -85,B 0,C 180,E1 -12681.762,E2 -12681.762} C_VEL
LIN {X 0,Y 367.566,Z 546.979,A -85,B 0,C 180,E1 -12683.413,E2 -12683.413} C_VEL
LIN {X 0,Y 367.466,Z 549.346,A -85,B 0,C 180,E1 -12684.513,E2 -12684.513} C_VEL
LIN {X 0,Y 367.438,Z 551.145,A -85,B 0,C 180,E1 -12685.612,E2 -12685.612} C_VEL
LIN {X 0,Y 367.36,Z 553.589,A -85,B 0,C 180,E1 -12687.807,E2 -12687.807} C_VEL
LIN {X 0,Y 367.403,Z 554.179,A -85,B 0,C 180,E1 -12688.904,E2 -12688.904} C_VEL
LIN {X 0,Y 367.403,Z 554.179,A -85,B 0,C 180,E1 -12691.096,E2 -12691.096} C_VEL
LIN {X 0,Y 367.36,Z 553.589,A -85,B 0,C 180,E1 -12692.193,E2 -12692.193} C_VEL
LIN {X 0,Y 367.438,Z 551.145,A -85,B 0,C 180,E1 -12694.388,E2 -12694.388} C_VEL
LIN {X 0,Y 367.48,Z 548.251,A -85,B 0,C 180,E1 -12696.012,E2 -12696.012} C_VEL
LIN {X 0,Y 367.726,Z 544.208,A -85,B 0,C 180,E1 -12697.688,E2 -12697.688} C_VEL
LIN {X 0,Y 368.115,Z 539.078,A -85,B 0,C 180,E1 -12699.339,E2 -12699.339} C_VEL
LIN {X 0,Y 368.614,Z 533.816,A -85,B 0,C 180,E1 -12700.713,E2 -12700.713} C_VEL
LIN {X 0,Y 369.255,Z 527.499,A -85,B 0,C 180,E1 -12702.085,E2 -12702.085} C_VEL
LIN {X 0,Y 369.94,Z 521.55,A -85,B 0,C 180,E1 -12703.177,E2 -12703.177} C_VEL
LIN {X 0,Y 370.577,Z 514.62,A -85,B 0,C 180,E1 -12704.273,E2 -12704.273} C_VEL
LIN {X 0,Y 371.392,Z 506.44,A -85,B 0,C 180,E1 -12705.362,E2 -12705.362} C_VEL
LIN {X 0,Y 372.234,Z 497.929,A -85,B 0,C 180,E1 -12706.31,E2 -12706.31} C_VEL
LIN {X 0,Y 373.046,Z 489.213,A -85,B 0,C 180,E1 -12707.119,E2 -12707.119} C_VEL
LIN {X 0,Y 373.943,Z 479.458,A -85,B 0,C 180,E1 -12707.853,E2 -12707.853} C_VEL
LIN {X 0,Y 374.511,Z 470.664,A -85,B 0,C 180,E1 -12708.391,E2 -12708.391} C_VEL
LIN {X 0,Y 375.195,Z 460.741,A -85,B 0,C 180,E1 -12708.851,E2 -12708.851} C_VEL
LIN {X 0,Y 375.622,Z 450.89,A -85,B 0,C 180,E1 -12709.183,E2 -12709.183} C_VEL
LIN {X 0,Y 376.054,Z 428.073,A -85,B 0,C 180,E1 -12709.657,E2 -12709.657} C_VEL
LIN {X 0,Y 376.707,Z 376.064,A -85,B 0,C 180,E1 -12710.655,E2 -12710.655} C_VEL
LIN {X 0,Y 371.37,Z 347.489,A -85,B 0,C 180,E1 -12711.543,E2 -12711.543} C_VEL
LIN {X 0,Y 370.57,Z 343.39,A -85,B 0,C 180,E1 -12711.72,E2 -12711.72} C_VEL
LIN {X 0,Y 371.819,Z 331.368,A -85,B 0,C 180,E1 -12715.209,E2 -12715.209} C_VEL
LIN {X 0,Y 371.875,Z 327.491,A -85,B 0,C 180,E1 -12716.366,E2 -12716.366} C_VEL
LIN {X 0,Y 370.238,Z 318.507,A -85,B 0,C 180,E1 -12719.168,E2 -12719.168} C_VEL
LIN {X 0,Y 368.926,Z 312.049,A -85,B 0,C 180,E1 -12721.351,E2 -12721.351} C_VEL
LIN {X 0,Y 368.928,Z 312.021,A -85,B 0,C 180,E1 -12725,E2 -12725} C_VEL
LIN {X 0,Y 368.877,Z 312.033,A -85,B 0,C 180,E1 -12728.633,E2 -12728.633} C_VEL
LIN {X 0,Y 368.87,Z 312.026,A -85,B 0,C 180,E1 -12732.007,E2 -12732.007} C_VEL
LIN {X 0,Y 368.877,Z 312.032,A -85,B 0,C 180,E1 -12735.175,E2 -12735.175} C_VEL
LIN {X 0,Y 368.88,Z 312.034,A -85,B 0,C 180,E1 -12738.176,E2 -12738.176} C_VEL
LIN {X 0,Y 368.903,Z 312.026,A -85,B 0,C 180,E1 -12741.359,E2 -12741.359} C_VEL
LIN {X 0,Y 368.926,Z 312.019,A -85,B 0,C 180,E1 -12745.145,E2 -12745.145} C_VEL
LIN {X 0,Y 368.925,Z 312.028,A -85,B 0,C 180,E1 -12749.045,E2 -12749.045} C_VEL
LIN {X 0,Y 368.957,Z 312.006,A -85,B 0,C 180,E1 -12752.795,E2 -12752.795} C_VEL
LIN {X 0,Y 368.927,Z 312.027,A -85,B 0,C 180,E1 -12756.116,E2 -12756.116} C_VEL
LIN {X 0,Y 368.93,Z 312.011,A -85,B 0,C 180,E1 -12759.946,E2 -12759.946} C_VEL
LIN {X 0,Y 368.969,Z 312.01,A -85,B 0,C 180,E1 -12763.398,E2 -12763.398} C_VEL
LIN {X 0,Y 369.051,Z 312.01,A -85,B 0,C 180,E1 -12766.789,E2 -12766.789} C_VEL
LIN {X 0,Y 369.06,Z 311.982,A -85,B 0,C 180,E1 -12770.131,E2 -12770.131} C_VEL
LIN {X 0,Y 369.193,Z 311.99,A -85,B 0,C 180,E1 -12773.441,E2 -12773.441} C_VEL
LIN {X 0,Y 369.31,Z 311.97,A -85,B 0,C 180,E1 -12777.818,E2 -12777.818} C_VEL
LIN {X 0,Y 369.449,Z 311.932,A -85,B 0,C 180,E1 -12779.999,E2 -12779.999} C_VEL
LIN {X 0,Y 369.308,Z 311.968,A -85,B 0,C 180,E1 -12782.181,E2 -12782.181} C_VEL
LIN {X 0,Y 369.185,Z 311.994,A -85,B 0,C 180,E1 -12786.627,E2 -12786.627} C_VEL
LIN {X 0,Y 369.059,Z 311.982,A -85,B 0,C 180,E1 -12789.868,E2 -12789.868} C_VEL
LIN {X 0,Y 369.028,Z 312.015,A -85,B 0,C 180,E1 -12793.772,E2 -12793.772} C_VEL
LIN {X 0,Y 368.993,Z 312.005,A -85,B 0,C 180,E1 -12797.768,E2 -12797.768} C_VEL
LIN {X 0,Y 368.921,Z 312.021,A -85,B 0,C 180,E1 -12801.219,E2 -12801.219} C_VEL
LIN {X 0,Y 368.949,Z 312.025,A -85,B 0,C 180,E1 -12804.775,E2 -12804.775} C_VEL
LIN {X 0,Y 368.978,Z 312.007,A -85,B 0,C 180,E1 -12808.435,E2 -12808.435} C_VEL
LIN {X 0,Y 368.894,Z 312.033,A -85,B 0,C 180,E1 -12812.238,E2 -12812.238} C_VEL
LIN {X 0,Y 368.921,Z 312.017,A -85,B 0,C 180,E1 -12815.002,E2 -12815.002} C_VEL
LIN {X 0,Y 368.905,Z 312.033,A -85,B 0,C 180,E1 -12818.641,E2 -12818.641} C_VEL
LIN {X 0,Y 368.934,Z 312.022,A -85,B 0,C 180,E1 -12822.02,E2 -12822.02} C_VEL
LIN {X 0,Y 368.917,Z 312.02,A -85,B 0,C 180,E1 -12825.183,E2 -12825.183} C_VEL
LIN {X 0,Y 368.887,Z 311.994,A -85,B 0,C 180,E1 -12828.179,E2 -12828.179} C_VEL
LIN {X 0,Y 368.906,Z 312.032,A -85,B 0,C 180,E1 -12831.359,E2 -12831.359} C_VEL
LIN {X 0,Y 368.93,Z 312.002,A -85,B 0,C 180,E1 -12835.147,E2 -12835.147} C_VEL
LIN {X 0,Y 368.923,Z 312.027,A -85,B 0,C 180,E1 -12839.047,E2 -12839.047} C_VEL
LIN {X 0,Y 368.957,Z 312.028,A -85,B 0,C 180,E1 -12842.797,E2 -12842.797} C_VEL
LIN {X 0,Y 368.94,Z 312.031,A -85,B 0,C 180,E1 -12846.113,E2 -12846.113} C_VEL
LIN {X 0,Y 368.932,Z 312.031,A -85,B 0,C 180,E1 -12849.947,E2 -12849.947} C_VEL
LIN {X 0,Y 368.971,Z 312.026,A -85,B 0,C 180,E1 -12853.399,E2 -12853.399} C_VEL
LIN {X 0,Y 369.036,Z 312.423,A -85,B 0,C 180,E1 -12854.112,E2 -12854.112} C_VEL
LIN {X 0,Y 369.45,Z 313.789,A -85,B 0,C 180,E1 -12854.431,E2 -12854.431} C_VEL
LIN {X 0,Y 370.843,Z 315.968,A -85,B 0,C 180,E1 -12854.93,E2 -12854.93} C_VEL
LIN {X 0,Y 373.91,Z 318.24,A -85,B 0,C 180,E1 -12855.94,E2 -12855.94} C_VEL
LIN {X 0,Y 375.803,Z 321.293,A -85,B 0,C 180,E1 -12856.694,E2 -12856.694} C_VEL
LIN {X 0,Y 378.433,Z 323.424,A -85,B 0,C 180,E1 -12857.669,E2 -12857.669} C_VEL
LIN {X 0,Y 379.535,Z 324.2,A -85,B 0,C 180,E1 -12858.132,E2 -12858.132} C_VEL
LIN {X 0,Y 381.399,Z 326.946,A -85,B 0,C 180,E1 -12858.979,E2 -12858.979} C_VEL
LIN {X 0,Y 384.05,Z 329.301,A -85,B 0,C 180,E1 -12860.26,E2 -12860.26} C_VEL
LIN {X 0,Y 386.289,Z 330.549,A -85,B 0,C 180,E1 -12861.434,E2 -12861.434} C_VEL
LIN {X 0,Y 388.224,Z 333.442,A -85,B 0,C 180,E1 -12862.72,E2 -12862.72} C_VEL
LIN {X 0,Y 390.286,Z 335.325,A -85,B 0,C 180,E1 -12864.316,E2 -12864.316} C_VEL
LIN {X 0,Y 391.884,Z 336.237,A -85,B 0,C 180,E1 -12865.886,E2 -12865.886} C_VEL
LIN {X 0,Y 392.994,Z 336.616,A -85,B 0,C 180,E1 -12867.456,E2 -12867.456} C_VEL
LIN {X 0,Y 393.545,Z 337.05,A -85,B 0,C 180,E1 -12868.977,E2 -12868.977} C_VEL
LIN {X 0,Y 393.727,Z 336.99,A -85,B 0,C 180,E1 -12870,E2 -12870} C_VEL
LIN {X 0,Y 393.467,Z 336.923,A -85,B 0,C 180,E1 -12871.535,E2 -12871.535} C_VEL
LIN {X 0,Y 392.738,Z 336.497,A -85,B 0,C 180,E1 -12873.077,E2 -12873.077} C_VEL
LIN {X 0,Y 391.175,Z 335.888,A -85,B 0,C 180,E1 -12874.895,E2 -12874.895} C_VEL
LIN {X 0,Y 389.129,Z 334.378,A -85,B 0,C 180,E1 -12876.619,E2 -12876.619} C_VEL
LIN {X 0,Y 387.297,Z 332.108,A -85,B 0,C 180,E1 -12877.941,E2 -12877.941} C_VEL
LIN {X 0,Y 385.95,Z 330.187,A -85,B 0,C 180,E1 -12878.772,E2 -12878.772} C_VEL
LIN {X 0,Y 383.231,Z 328.735,A -85,B 0,C 180,E1 -12880.134,E2 -12880.134} C_VEL
LIN {X 0,Y 380.894,Z 326.366,A -85,B 0,C 180,E1 -12881.238,E2 -12881.238} C_VEL
LIN {X 0,Y 379.161,Z 323.789,A -85,B 0,C 180,E1 -12882.036,E2 -12882.036} C_VEL
LIN {X 0,Y 376.571,Z 322.101,A -85,B 0,C 180,E1 -12883.011,E2 -12883.011} C_VEL
LIN {X 0,Y 374.518,Z 319.355,A -85,B 0,C 180,E1 -12883.833,E2 -12883.833} C_VEL
LIN {X 0,Y 373.643,Z 317.888,A -85,B 0,C 180,E1 -12884.153,E2 -12884.153} C_VEL
LIN {X 0,Y 370.851,Z 315.972,A -85,B 0,C 180,E1 -12885.068,E2 -12885.068} C_VEL
LIN {X 0,Y 369.451,Z 313.791,A -85,B 0,C 180,E1 -12885.569,E2 -12885.569} C_VEL
LIN {X 0,Y 369.036,Z 312.425,A -85,B 0,C 180,E1 -12885.888,E2 -12885.888} C_VEL
LIN {X 0,Y 368.971,Z 312.026,A -85,B 0,C 180,E1 -12886.601,E2 -12886.601} C_VEL
LIN {X 0,Y 368.932,Z 312.032,A -85,B 0,C 180,E1 -12890.053,E2 -12890.053} C_VEL
LIN {X 0,Y 368.94,Z 312.031,A -85,B 0,C 180,E1 -12893.887,E2 -12893.887} C_VEL
LIN {X 0,Y 368.957,Z 312.028,A -85,B 0,C 180,E1 -12897.203,E2 -12897.203} C_VEL
LIN {X 0,Y 368.923,Z 312.027,A -85,B 0,C 180,E1 -12900.953,E2 -12900.953} C_VEL
LIN {X 0,Y 368.923,Z 312.003,A -85,B 0,C 180,E1 -12905.001,E2 -12905.001} C_VEL
LIN {X 0,Y 368.906,Z 312.032,A -85,B 0,C 180,E1 -12908.641,E2 -12908.641} C_VEL
LIN {X 0,Y 368.887,Z 311.994,A -85,B 0,C 180,E1 -12911.821,E2 -12911.821} C_VEL
LIN {X 0,Y 368.913,Z 312.02,A -85,B 0,C 180,E1 -12914.778,E2 -12914.778} C_VEL
LIN {X 0,Y 368.313,Z 312.108,A -85,B 0,C 180,E1 -12915.689,E2 -12915.689} C_VEL
LIN {X 0,Y 365.482,Z 312.461,A -85,B 0,C 180,E1 -12917.171,E2 -12917.171} C_VEL
LIN {X 0,Y 363.035,Z 312.756,A -85,B 0,C 180,E1 -12918.369,E2 -12918.369} C_VEL
LIN {X 0,Y 361.969,Z 312.885,A -85,B 0,C 180,E1 -12919.296,E2 -12919.296} C_VEL
LIN {X 0,Y 361.876,Z 312.897,A -85,B 0,C 180,E1 -12919.61,E2 -12919.61} C_VEL
LIN {X 0,Y 361.861,Z 312.912,A -85,B 0,C 180,E1 -12922.982,E2 -12922.982} C_VEL
LIN {X 0,Y 361.853,Z 312.9,A -85,B 0,C 180,E1 -12926.63,E2 -12926.63} C_VEL
LIN {X 0,Y 361.868,Z 312.907,A -85,B 0,C 180,E1 -12929.672,E2 -12929.672} C_VEL
LIN {X 0,Y 361.946,Z 312.883,A -85,B 0,C 180,E1 -12933.475,E2 -12933.475} C_VEL
LIN {X 0,Y 361.883,Z 312.908,A -85,B 0,C 180,E1 -12937.145,E2 -12937.145} C_VEL
LIN {X 0,Y 361.903,Z 312.88,A -85,B 0,C 180,E1 -12940.724,E2 -12940.724} C_VEL
LIN {X 0,Y 361.924,Z 312.892,A -85,B 0,C 180,E1 -12943.066,E2 -12943.066} C_VEL
LIN {X 0,Y 361.99,Z 312.893,A -85,B 0,C 180,E1 -12946.528,E2 -12946.528} C_VEL
LIN {X 0,Y 362.023,Z 312.857,A -85,B 0,C 180,E1 -12949.938,E2 -12949.938} C_VEL
LIN {X 0,Y 362.154,Z 312.872,A -85,B 0,C 180,E1 -12953.314,E2 -12953.314} C_VEL
LIN {X 0,Y 362.272,Z 312.844,A -85,B 0,C 180,E1 -12957.777,E2 -12957.777} C_VEL
LIN {X 0,Y 362.419,Z 312.807,A -85,B 0,C 180,E1 -12960.001,E2 -12960.001} C_VEL
LIN {X 0,Y 362.274,Z 312.847,A -85,B 0,C 180,E1 -12962.224,E2 -12962.224} C_VEL
LIN {X 0,Y 362.154,Z 312.865,A -85,B 0,C 180,E1 -12966.687,E2 -12966.687} C_VEL
LIN {X 0,Y 362.024,Z 312.858,A -85,B 0,C 180,E1 -12970.063,E2 -12970.063} C_VEL
LIN {X 0,Y 361.991,Z 312.89,A -85,B 0,C 180,E1 -12973.899,E2 -12973.899} C_VEL
LIN {X 0,Y 361.961,Z 312.873,A -85,B 0,C 180,E1 -12977.939,E2 -12977.939} C_VEL
LIN {X 0,Y 361.855,Z 312.904,A -85,B 0,C 180,E1 -12981.656,E2 -12981.656} C_VEL
LIN {X 0,Y 361.92,Z 312.889,A -85,B 0,C 180,E1 -12985.291,E2 -12985.291} C_VEL
LIN {X 0,Y 361.903,Z 312.887,A -85,B 0,C 180,E1 -12987.78,E2 -12987.78} C_VEL
LIN {X 0,Y 361.833,Z 312.911,A -85,B 0,C 180,E1 -12991.631,E2 -12991.631} C_VEL
LIN {X 0,Y 361.866,Z 312.901,A -85,B 0,C 180,E1 -12995.345,E2 -12995.345} C_VEL
LIN {X 0,Y 361.864,Z 312.901,A -85,B 0,C 180,E1 -12999.027,E2 -12999.027} C_VEL
LIN {X 0,Y 361.833,Z 312.911,A -85,B 0,C 180,E1 -13002.83,E2 -13002.83} C_VEL
LIN {X 0,Y 361.816,Z 312.916,A -85,B 0,C 180,E1 -13005.948,E2 -13005.948} C_VEL
LIN {X 0,Y 361.811,Z 312.893,A -85,B 0,C 180,E1 -13009.25,E2 -13009.25} C_VEL
LIN {X 0,Y 361.864,Z 312.906,A -85,B 0,C 180,E1 -13012.983,E2 -13012.983} C_VEL
LIN {X 0,Y 361.859,Z 312.907,A -85,B 0,C 180,E1 -13016.632,E2 -13016.632} C_VEL
LIN {X 0,Y 361.927,Z 313.033,A -85,B 0,C 180,E1 -13018.38,E2 -13018.38} C_VEL
LIN {X 0,Y 363.467,Z 320.815,A -85,B 0,C 180,E1 -13021.093,E2 -13021.093} C_VEL
LIN {X 0,Y 364.941,Z 329.18,A -85,B 0,C 180,E1 -13023.71,E2 -13023.71} C_VEL
LIN {X 0,Y 364.752,Z 333.315,A -85,B 0,C 180,E1 -13024.92,E2 -13024.92} C_VEL
LIN {X 0,Y 363.68,Z 343.176,A -85,B 0,C 180,E1 -13027.844,E2 -13027.844} C_VEL
LIN {X 0,Y 364.854,Z 349.106,A -85,B 0,C 180,E1 -13028.09,E2 -13028.09} C_VEL
LIN {X 0,Y 369.924,Z 376.265,A -85,B 0,C 180,E1 -13028.956,E2 -13028.956} C_VEL
LIN {X 0,Y 370.161,Z 381.939,A -85,B 0,C 180,E1 -13029.086,E2 -13029.086} C_VEL
LIN {X 0,Y 368.992,Z 449.365,A -85,B 0,C 180,E1 -13030.422,E2 -13030.422} C_VEL
LIN {X 0,Y 368.535,Z 459.673,A -85,B 0,C 180,E1 -13030.759,E2 -13030.759} C_VEL
LIN {X 0,Y 367.884,Z 469.183,A -85,B 0,C 180,E1 -13031.194,E2 -13031.194} C_VEL
LIN {X 0,Y 367.214,Z 478.256,A -85,B 0,C 180,E1 -13031.736,E2 -13031.736} C_VEL
LIN {X 0,Y 366.415,Z 487.388,A -85,B 0,C 180,E1 -13032.417,E2 -13032.417} C_VEL
LIN {X 0,Y 365.573,Z 496.384,A -85,B 0,C 180,E1 -13033.24,E2 -13033.24} C_VEL
LIN {X 0,Y 364.645,Z 505.11,A -85,B 0,C 180,E1 -13034.203,E2 -13034.203} C_VEL
LIN {X 0,Y 363.848,Z 513.033,A -85,B 0,C 180,E1 -13035.25,E2 -13035.25} C_VEL
LIN {X 0,Y 362.97,Z 521.354,A -85,B 0,C 180,E1 -13036.565,E2 -13036.565} C_VEL
LIN {X 0,Y 362.282,Z 527.304,A -85,B 0,C 180,E1 -13037.679,E2 -13037.679} C_VEL
LIN {X 0,Y 361.593,Z 533.621,A -85,B 0,C 180,E1 -13039.076,E2 -13039.076} C_VEL
LIN {X 0,Y 361.068,Z 538.883,A -85,B 0,C 180,E1 -13040.477,E2 -13040.477} C_VEL
LIN {X 0,Y 360.676,Z 544.013,A -85,B 0,C 180,E1 -13042.161,E2 -13042.161} C_VEL
LIN {X 0,Y 360.413,Z 548.314,A -85,B 0,C 180,E1 -13043.988,E2 -13043.988} C_VEL
LIN {X 0,Y 360.349,Z 550.951,A -85,B 0,C 180,E1 -13045.526,E2 -13045.526} C_VEL
LIN {X 0,Y 360.264,Z 553.395,A -85,B 0,C 180,E1 -13047.764,E2 -13047.764} C_VEL
LIN {X 0,Y 360.303,Z 553.985,A -85,B 0,C 180,E1 -13048.882,E2 -13048.882} C_VEL
LIN {X 0,Y 360.303,Z 553.985,A -85,B 0,C 180,E1 -13051.118,E2 -13051.118} C_VEL
LIN {X 0,Y 360.264,Z 553.395,A -85,B 0,C 180,E1 -13052.236,E2 -13052.236} C_VEL
LIN {X 0,Y 360.349,Z 550.951,A -85,B 0,C 180,E1 -13054.474,E2 -13054.474} C_VEL
LIN {X 0,Y 360.379,Z 548.426,A -85,B 0,C 180,E1 -13055.961,E2 -13055.961} C_VEL
LIN {X 0,Y 360.594,Z 545.544,A -85,B 0,C 180,E1 -13057.278,E2 -13057.278} C_VEL
LIN {X 0,Y 360.933,Z 540.799,A -85,B 0,C 180,E1 -13058.961,E2 -13058.961} C_VEL
LIN {X 0,Y 361.511,Z 534.777,A -85,B 0,C 180,E1 -13060.643,E2 -13060.643} C_VEL
LIN {X 0,Y 362.107,Z 528.68,A -85,B 0,C 180,E1 -13062.043,E2 -13062.043} C_VEL
LIN {X 0,Y 362.815,Z 522.982,A -85,B 0,C 180,E1 -13063.156,E2 -13063.156} C_VEL
LIN {X 0,Y 363.685,Z 514.426,A -85,B 0,C 180,E1 -13064.549,E2 -13064.549} C_VEL
LIN {X 0,Y 364.527,Z 506.245,A -85,B 0,C 180,E1 -13065.659,E2 -13065.659} C_VEL
LIN {X 0,Y 365.422,Z 497.735,A -85,B 0,C 180,E1 -13066.623,E2 -13066.623} C_VEL
LIN {X 0,Y 366.268,Z 489.019,A -85,B 0,C 180,E1 -13067.446,E2 -13067.446} C_VEL
LIN {X 0,Y 367.178,Z 479.264,A -85,B 0,C 180,E1 -13068.193,E2 -13068.193} C_VEL
LIN {X 0,Y 367.767,Z 470.469,A -85,B 0,C 180,E1 -13068.74,E2 -13068.74} C_VEL
LIN {X 0,Y 368.485,Z 460.547,A -85,B 0,C 180,E1 -13069.208,E2 -13069.208} C_VEL
LIN {X 0,Y 368.943,Z 450.696,A -85,B 0,C 180,E1 -13069.545,E2 -13069.545} C_VEL
LIN {X 0,Y 369.376,Z 427.879,A -85,B 0,C 180,E1 -13070.028,E2 -13070.028} C_VEL
LIN {X 0,Y 370.109,Z 377.161,A -85,B 0,C 180,E1 -13071.015,E2 -13071.015} C_VEL
LIN {X 0,Y 364.799,Z 348.826,A -85,B 0,C 180,E1 -13071.919,E2 -13071.919} C_VEL
LIN {X 0,Y 363.697,Z 343.452,A -85,B 0,C 180,E1 -13072.126,E2 -13072.126} C_VEL
LIN {X 0,Y 363.683,Z 342.738,A -85,B 0,C 180,E1 -13072.238,E2 -13072.238} C_VEL
LIN {X 0,Y 364.987,Z 331.321,A -85,B 0,C 180,E1 -13075.673,E2 -13075.673} C_VEL
LIN {X 0,Y 364.734,Z 327.446,A -85,B 0,C 180,E1 -13076.877,E2 -13076.877} C_VEL
LIN {X 0,Y 363.007,Z 318.459,A -85,B 0,C 180,E1 -13079.766,E2 -13079.766} C_VEL
LIN {X 0,Y 361.911,Z 313.003,A -85,B 0,C 180,E1 -13081.621,E2 -13081.621} C_VEL
LIN {X 0,Y 361.867,Z 312.896,A -85,B 0,C 180,E1 -13085.636,E2 -13085.636} C_VEL
LIN {X 0,Y 361.826,Z 312.907,A -85,B 0,C 180,E1 -13089.017,E2 -13089.017} C_VEL
LIN {X 0,Y 361.832,Z 312.912,A -85,B 0,C 180,E1 -13092.828,E2 -13092.828} C_VEL
LIN {X 0,Y 361.815,Z 312.91,A -85,B 0,C 180,E1 -13095.946,E2 -13095.946} C_VEL
LIN {X 0,Y 361.832,Z 312.908,A -85,B 0,C 180,E1 -13099.244,E2 -13099.244} C_VEL
LIN {X 0,Y 361.857,Z 312.909,A -85,B 0,C 180,E1 -13102.777,E2 -13102.777} C_VEL
LIN {X 0,Y 361.846,Z 312.896,A -85,B 0,C 180,E1 -13105.718,E2 -13105.718} C_VEL
LIN {X 0,Y 361.868,Z 312.911,A -85,B 0,C 180,E1 -13109.671,E2 -13109.671} C_VEL
LIN {X 0,Y 361.948,Z 312.877,A -85,B 0,C 180,E1 -13113.474,E2 -13113.474} C_VEL
LIN {X 0,Y 361.873,Z 312.907,A -85,B 0,C 180,E1 -13117.143,E2 -13117.143} C_VEL
LIN {X 0,Y 361.9,Z 312.882,A -85,B 0,C 180,E1 -13120.722,E2 -13120.722} C_VEL
LIN {X 0,Y 361.926,Z 312.883,A -85,B 0,C 180,E1 -13123.065,E2 -13123.065} C_VEL
LIN {X 0,Y 361.992,Z 312.889,A -85,B 0,C 180,E1 -13126.527,E2 -13126.527} C_VEL
LIN {X 0,Y 362.024,Z 312.858,A -85,B 0,C 180,E1 -13129.937,E2 -13129.937} C_VEL
LIN {X 0,Y 362.154,Z 312.865,A -85,B 0,C 180,E1 -13133.313,E2 -13133.313} C_VEL
LIN {X 0,Y 362.274,Z 312.847,A -85,B 0,C 180,E1 -13137.776,E2 -13137.776} C_VEL
LIN {X 0,Y 362.419,Z 312.807,A -85,B 0,C 180,E1 -13139.999,E2 -13139.999} C_VEL
LIN {X 0,Y 362.272,Z 312.844,A -85,B 0,C 180,E1 -13142.223,E2 -13142.223} C_VEL
LIN {X 0,Y 362.154,Z 312.872,A -85,B 0,C 180,E1 -13146.686,E2 -13146.686} C_VEL
LIN {X 0,Y 362.023,Z 312.857,A -85,B 0,C 180,E1 -13150.062,E2 -13150.062} C_VEL
LIN {X 0,Y 361.989,Z 312.891,A -85,B 0,C 180,E1 -13153.898,E2 -13153.898} C_VEL
LIN {X 0,Y 361.959,Z 312.881,A -85,B 0,C 180,E1 -13157.938,E2 -13157.938} C_VEL
LIN {X 0,Y 361.885,Z 312.902,A -85,B 0,C 180,E1 -13161.653,E2 -13161.653} C_VEL
LIN {X 0,Y 361.919,Z 312.894,A -85,B 0,C 180,E1 -13165.29,E2 -13165.29} C_VEL
LIN {X 0,Y 361.914,Z 312.883,A -85,B 0,C 180,E1 -13167.778,E2 -13167.778} C_VEL
LIN {X 0,Y 361.839,Z 312.913,A -85,B 0,C 180,E1 -13171.285,E2 -13171.285} C_VEL
LIN {X 0,Y 361.847,Z 312.897,A -85,B 0,C 180,E1 -13174.28,E2 -13174.28} C_VEL
LIN {X 0,Y 361.858,Z 312.911,A -85,B 0,C 180,E1 -13177.223,E2 -13177.223} C_VEL
LIN {X 0,Y 361.897,Z 312.894,A -85,B 0,C 180,E1 -13180.768,E2 -13180.768} C_VEL
LIN {X 0,Y 361.897,Z 312.904,A -85,B 0,C 180,E1 -13184.355,E2 -13184.355} C_VEL
LIN {X 0,Y 361.835,Z 312.871,A -85,B 0,C 180,E1 -13187.567,E2 -13187.567} C_VEL
LIN {X 0,Y 361.868,Z 312.906,A -85,B 0,C 180,E1 -13190.973,E2 -13190.973} C_VEL
LIN {X 0,Y 361.868,Z 312.884,A -85,B 0,C 180,E1 -13194.655,E2 -13194.655} C_VEL
LIN {X 0,Y 361.832,Z 312.917,A -85,B 0,C 180,E1 -13198.371,E2 -13198.371} C_VEL
LIN {X 0,Y 361.903,Z 312.901,A -85,B 0,C 180,E1 -13202.221,E2 -13202.221} C_VEL
LIN {X 0,Y 361.923,Z 312.904,A -85,B 0,C 180,E1 -13204.71,E2 -13204.71} C_VEL
LIN {X 0,Y 361.887,Z 312.909,A -85,B 0,C 180,E1 -13208.347,E2 -13208.347} C_VEL
LIN {X 0,Y 361.958,Z 313.007,A -85,B 0,C 180,E1 -13212.141,E2 -13212.141} C_VEL
LIN {X 0,Y 362.155,Z 313.99,A -85,B 0,C 180,E1 -13212.511,E2 -13212.511} C_VEL
LIN {X 0,Y 363.707,Z 316.778,A -85,B 0,C 180,E1 -13213.03,E2 -13213.03} C_VEL
LIN {X 0,Y 366.071,Z 318.534,A -85,B 0,C 180,E1 -13213.721,E2 -13213.721} C_VEL
LIN {X 0,Y 368.394,Z 321.975,A -85,B 0,C 180,E1 -13214.471,E2 -13214.471} C_VEL
LIN {X 0,Y 371.016,Z 324.158,A -85,B 0,C 180,E1 -13215.324,E2 -13215.324} C_VEL
LIN {X 0,Y 371.855,Z 324.832,A -85,B 0,C 180,E1 -13215.602,E2 -13215.602} C_VEL
LIN {X 0,Y 374.175,Z 328.04,A -85,B 0,C 180,E1 -13216.445,E2 -13216.445} C_VEL
LIN {X 0,Y 376.963,Z 330.265,A -85,B 0,C 180,E1 -13217.483,E2 -13217.483} C_VEL
LIN {X 0,Y 377.932,Z 331.029,A -85,B 0,C 180,E1 -13217.856,E2 -13217.856} C_VEL
LIN {X 0,Y 380.36,Z 334.213,A -85,B 0,C 180,E1 -13218.948,E2 -13218.948} C_VEL
LIN {X 0,Y 383.08,Z 336.367,A -85,B 0,C 180,E1 -13220.235,E2 -13220.235} C_VEL
LIN {X 0,Y 384.988,Z 337.45,A -85,B 0,C 180,E1 -13221.206,E2 -13221.206} C_VEL
LIN {X 0,Y 387.164,Z 340.429,A -85,B 0,C 180,E1 -13222.596,E2 -13222.596} C_VEL
LIN {X 0,Y 389.397,Z 342.369,A -85,B 0,C 180,E1 -13224.303,E2 -13224.303} C_VEL
LIN {X 0,Y 391.009,Z 343.283,A -85,B 0,C 180,E1 -13225.877,E2 -13225.877} C_VEL
LIN {X 0,Y 392.127,Z 343.664,A -85,B 0,C 180,E1 -13227.451,E2 -13227.451} C_VEL
LIN {X 0,Y 392.684,Z 344.085,A -85,B 0,C 180,E1 -13228.975,E2 -13228.975} C_VEL
LIN {X 0,Y 392.864,Z 344.022,A -85,B 0,C 180,E1 -13230,E2 -13230} C_VEL
LIN {X 0,Y 392.598,Z 343.971,A -85,B 0,C 180,E1 -13231.539,E2 -13231.539} C_VEL
LIN {X 0,Y 391.863,Z 343.543,A -85,B 0,C 180,E1 -13233.084,E2 -13233.084} C_VEL
LIN {X 0,Y 390.285,Z 342.933,A -85,B 0,C 180,E1 -13234.907,E2 -13234.907} C_VEL
LIN {X 0,Y 388.217,Z 341.449,A -85,B 0,C 180,E1 -13236.635,E2 -13236.635} C_VEL
LIN {X 0,Y 386.33,Z 339.399,A -85,B 0,C 180,E1 -13237.961,E2 -13237.961} C_VEL
LIN {X 0,Y 384.775,Z 337.129,A -85,B 0,C 180,E1 -13238.931,E2 -13238.931} C_VEL
LIN {X 0,Y 381.794,Z 335.491,A -85,B 0,C 180,E1 -13240.39,E2 -13240.39} C_VEL
LIN {X 0,Y 379.123,Z 332.823,A -85,B 0,C 180,E1 -13241.589,E2 -13241.589} C_VEL
LIN {X 0,Y 377.388,Z 330.465,A -85,B 0,C 180,E1 -13242.366,E2 -13242.366} C_VEL
LIN {X 0,Y 374.536,Z 328.422,A -85,B 0,C 180,E1 -13243.414,E2 -13243.414} C_VEL
LIN {X 0,Y 372.28,Z 325.518,A -85,B 0,C 180,E1 -13244.244,E2 -13244.244} C_VEL
LIN {X 0,Y 371.416,Z 324.377,A -85,B 0,C 180,E1 -13244.548,E2 -13244.548} C_VEL
LIN {X 0,Y 368.653,Z 322.236,A -85,B 0,C 180,E1 -13245.452,E2 -13245.452} C_VEL
LIN {X 0,Y 366.787,Z 319.684,A -85,B 0,C 180,E1 -13246.042,E2 -13246.042} C_VEL
LIN {X 0,Y 366.071,Z 318.534,A -85,B 0,C 180,E1 -13246.279,E2 -13246.279} C_VEL
LIN {X 0,Y 363.706,Z 316.778,A -85,B 0,C 180,E1 -13246.97,E2 -13246.97} C_VEL
LIN {X 0,Y 362.154,Z 313.987,A -85,B 0,C 180,E1 -13247.489,E2 -13247.489} C_VEL
LIN {X 0,Y 361.959,Z 313.007,A -85,B 0,C 180,E1 -13247.859,E2 -13247.859} C_VEL
LIN {X 0,Y 361.887,Z 312.909,A -85,B 0,C 180,E1 -13251.653,E2 -13251.653} C_VEL
LIN {X 0,Y 361.923,Z 312.904,A -85,B 0,C 180,E1 -13255.29,E2 -13255.29} C_VEL
LIN {X 0,Y 361.903,Z 312.901,A -85,B 0,C 180,E1 -13257.779,E2 -13257.779} C_VEL
LIN {X 0,Y 361.832,Z 312.917,A -85,B 0,C 180,E1 -13261.629,E2 -13261.629} C_VEL
LIN {X 0,Y 361.868,Z 312.884,A -85,B 0,C 180,E1 -13265.345,E2 -13265.345} C_VEL
LIN {X 0,Y 361.868,Z 312.906,A -85,B 0,C 180,E1 -13269.027,E2 -13269.027} C_VEL
LIN {X 0,Y 361.835,Z 312.871,A -85,B 0,C 180,E1 -13272.433,E2 -13272.433} C_VEL
LIN {X 0,Y 361.891,Z 312.906,A -85,B 0,C 180,E1 -13275.933,E2 -13275.933} C_VEL
LIN {X 0,Y 361.876,Z 312.897,A -85,B 0,C 180,E1 -13279.61,E2 -13279.61} C_VEL
LIN {X 0,Y 361.195,Z 312.987,A -85,B 0,C 180,E1 -13280.538,E2 -13280.538} C_VEL
LIN {X 0,Y 358.343,Z 313.348,A -85,B 0,C 180,E1 -13282.048,E2 -13282.048} C_VEL
LIN {X 0,Y 355.933,Z 313.647,A -85,B 0,C 180,E1 -13283.27,E2 -13283.27} C_VEL
LIN {X 0,Y 354.893,Z 313.77,A -85,B 0,C 180,E1 -13284.214,E2 -13284.214} C_VEL
LIN {X 0,Y 354.805,Z 313.778,A -85,B 0,C 180,E1 -13284.534,E2 -13284.534} C_VEL
LIN {X 0,Y 354.781,Z 313.792,A -85,B 0,C 180,E1 -13287.667,E2 -13287.667} C_VEL
LIN {X 0,Y 354.861,Z 313.778,A -85,B 0,C 180,E1 -13290.621,E2 -13290.621} C_VEL
LIN {X 0,Y 354.891,Z 313.767,A -85,B 0,C 180,E1 -13294.173,E2 -13294.173} C_VEL
LIN {X 0,Y 354.827,Z 313.781,A -85,B 0,C 180,E1 -13297.894,E2 -13297.894} C_VEL
LIN {X 0,Y 354.914,Z 313.757,A -85,B 0,C 180,E1 -13301.892,E2 -13301.892} C_VEL
LIN {X 0,Y 354.934,Z 313.77,A -85,B 0,C 180,E1 -13305.982,E2 -13305.982} C_VEL
LIN {X 0,Y 354.969,Z 313.736,A -85,B 0,C 180,E1 -13309.736,E2 -13309.736} C_VEL
LIN {X 0,Y 355.117,Z 313.747,A -85,B 0,C 180,E1 -13313.181,E2 -13313.181} C_VEL
LIN {X 0,Y 355.235,Z 313.72,A -85,B 0,C 180,E1 -13317.733,E2 -13317.733} C_VEL
LIN {X 0,Y 355.368,Z 313.685,A -85,B 0,C 180,E1 -13320.001,E2 -13320.001} C_VEL
LIN {X 0,Y 355.237,Z 313.723,A -85,B 0,C 180,E1 -13322.268,E2 -13322.268} C_VEL
LIN {X 0,Y 355.118,Z 313.739,A -85,B 0,C 180,E1 -13326.82,E2 -13326.82} C_VEL
LIN {X 0,Y 354.971,Z 313.737,A -85,B 0,C 180,E1 -13330.265,E2 -13330.265} C_VEL
LIN {X 0,Y 354.936,Z 313.769,A -85,B 0,C 180,E1 -13334.019,E2 -13334.019} C_VEL
LIN {X 0,Y 354.916,Z 313.749,A -85,B 0,C 180,E1 -13338.109,E2 -13338.109} C_VEL
LIN {X 0,Y 354.809,Z 313.784,A -85,B 0,C 180,E1 -13342.108,E2 -13342.108} C_VEL
LIN {X 0,Y 354.892,Z 313.761,A -85,B 0,C 180,E1 -13345.829,E2 -13345.829} C_VEL
LIN {X 0,Y 354.813,Z 313.784,A -85,B 0,C 180,E1 -13349.683,E2 -13349.683} C_VEL
LIN {X 0,Y 354.802,Z 313.773,A -85,B 0,C 180,E1 -13353.703,E2 -13353.703} C_VEL
LIN {X 0,Y 354.791,Z 313.791,A -85,B 0,C 180,E1 -13356.461,E2 -13356.461} C_VEL
LIN {X 0,Y 354.821,Z 313.777,A -85,B 0,C 180,E1 -13359.425,E2 -13359.425} C_VEL
LIN {X 0,Y 354.785,Z 313.789,A -85,B 0,C 180,E1 -13362.868,E2 -13362.868} C_VEL
LIN {X 0,Y 354.765,Z 313.796,A -85,B 0,C 180,E1 -13366.105,E2 -13366.105} C_VEL
LIN {X 0,Y 354.764,Z 313.77,A -85,B 0,C 180,E1 -13369.177,E2 -13369.177} C_VEL
LIN {X 0,Y 354.8,Z 313.789,A -85,B 0,C 180,E1 -13372.405,E2 -13372.405} C_VEL
LIN {X 0,Y 354.811,Z 313.778,A -85,B 0,C 180,E1 -13374.942,E2 -13374.942} C_VEL
LIN {X 0,Y 354.861,Z 313.85,A -85,B 0,C 180,E1 -13377.978,E2 -13377.978} C_VEL
LIN {X 0,Y 356.414,Z 321.673,A -85,B 0,C 180,E1 -13380.789,E2 -13380.789} C_VEL
LIN {X 0,Y 357.928,Z 330.042,A -85,B 0,C 180,E1 -13383.468,E2 -13383.468} C_VEL
LIN {X 0,Y 357.881,Z 333.742,A -85,B 0,C 180,E1 -13384.602,E2 -13384.602} C_VEL
LIN {X 0,Y 356.815,Z 342.961,A -85,B 0,C 180,E1 -13387.391,E2 -13387.391} C_VEL
LIN {X 0,Y 357.939,Z 348.525,A -85,B 0,C 180,E1 -13387.636,E2 -13387.636} C_VEL
LIN {X 0,Y 363.238,Z 376.81,A -85,B 0,C 180,E1 -13388.565,E2 -13388.565} C_VEL
LIN {X 0,Y 363.54,Z 382.144,A -85,B 0,C 180,E1 -13388.695,E2 -13388.695} C_VEL
LIN {X 0,Y 362.324,Z 449.172,A -85,B 0,C 180,E1 -13390.046,E2 -13390.046} C_VEL
LIN {X 0,Y 361.848,Z 459.479,A -85,B 0,C 180,E1 -13390.389,E2 -13390.389} C_VEL
LIN {X 0,Y 361.187,Z 468.989,A -85,B 0,C 180,E1 -13390.832,E2 -13390.832} C_VEL
LIN {X 0,Y 360.466,Z 478.061,A -85,B 0,C 180,E1 -13391.382,E2 -13391.382} C_VEL
LIN {X 0,Y 359.639,Z 487.193,A -85,B 0,C 180,E1 -13392.075,E2 -13392.075} C_VEL
LIN {X 0,Y 358.739,Z 496.189,A -85,B 0,C 180,E1 -13392.911,E2 -13392.911} C_VEL
LIN {X 0,Y 357.799,Z 504.916,A -85,B 0,C 180,E1 -13393.892,E2 -13393.892} C_VEL
LIN {X 0,Y 357.024,Z 512.286,A -85,B 0,C 180,E1 -13394.877,E2 -13394.877} C_VEL
LIN {X 0,Y 356.22,Z 519.532,A -85,B 0,C 180,E1 -13396.014,E2 -13396.014} C_VEL
LIN {X 0,Y 355.513,Z 525.734,A -85,B 0,C 180,E1 -13397.15,E2 -13397.15} C_VEL
LIN {X 0,Y 354.687,Z 532.269,A -85,B 0,C 180,E1 -13398.572,E2 -13398.572} C_VEL
LIN {X 0,Y 354.258,Z 536.773,A -85,B 0,C 180,E1 -13399.715,E2 -13399.715} C_VEL
LIN {X 0,Y 353.738,Z 542.265,A -85,B 0,C 180,E1 -13401.431,E2 -13401.431} C_VEL
LIN {X 0,Y 353.419,Z 546.59,A -85,B 0,C 180,E1 -13403.148,E2 -13403.148} C_VEL
LIN {X 0,Y 353.291,Z 548.957,A -85,B 0,C 180,E1 -13404.292,E2 -13404.292} C_VEL
LIN {X 0,Y 353.264,Z 550.757,A -85,B 0,C 180,E1 -13405.436,E2 -13405.436} C_VEL
LIN {X 0,Y 353.173,Z 553.202,A -85,B 0,C 180,E1 -13407.719,E2 -13407.719} C_VEL
LIN {X 0,Y 353.203,Z 553.791,A -85,B 0,C 180,E1 -13408.86,E2 -13408.86} C_VEL
LIN {X 0,Y 353.203,Z 553.791,A -85,B 0,C 180,E1 -13411.14,E2 -13411.14} C_VEL
LIN {X 0,Y 353.173,Z 553.202,A -85,B 0,C 180,E1 -13412.281,E2 -13412.281} C_VEL
LIN {X 0,Y 353.264,Z 550.757,A -85,B 0,C 180,E1 -13414.564,E2 -13414.564} C_VEL
LIN {X 0,Y 353.298,Z 548.536,A -85,B 0,C 180,E1 -13415.937,E2 -13415.937} C_VEL
LIN {X 0,Y 353.517,Z 545.349,A -85,B 0,C 180,E1 -13417.424,E2 -13417.424} C_VEL
LIN {X 0,Y 353.887,Z 540.604,A -85,B 0,C 180,E1 -13419.141,E2 -13419.141} C_VEL
LIN {X 0,Y 354.478,Z 534.582,A -85,B 0,C 180,E1 -13420.856,E2 -13420.856} C_VEL
LIN {X 0,Y 355.146,Z 528.485,A -85,B 0,C 180,E1 -13422.282,E2 -13422.282} C_VEL
LIN {X 0,Y 355.886,Z 522.787,A -85,B 0,C 180,E1 -13423.417,E2 -13423.417} C_VEL
LIN {X 0,Y 356.802,Z 514.231,A -85,B 0,C 180,E1 -13424.836,E2 -13424.836} C_VEL
LIN {X 0,Y 357.675,Z 506.051,A -85,B 0,C 180,E1 -13425.967,E2 -13425.967} C_VEL
LIN {X 0,Y 358.621,Z 497.541,A -85,B 0,C 180,E1 -13426.948,E2 -13426.948} C_VEL
LIN {X 0,Y 359.505,Z 488.826,A -85,B 0,C 180,E1 -13427.785,E2 -13427.785} C_VEL
LIN {X 0,Y 360.434,Z 479.07,A -85,B 0,C 180,E1 -13428.546,E2 -13428.546} C_VEL
LIN {X 0,Y 361.052,Z 470.275,A -85,B 0,C 180,E1 -13429.102,E2 -13429.102} C_VEL
LIN {X 0,Y 361.774,Z 460.352,A -85,B 0,C 180,E1 -13429.579,E2 -13429.579} C_VEL
LIN {X 0,Y 362.279,Z 450.503,A -85,B 0,C 180,E1 -13429.919,E2 -13429.919} C_VEL
LIN {X 0,Y 362.719,Z 426.517,A -85,B 0,C 180,E1 -13430.435,E2 -13430.435} C_VEL
LIN {X 0,Y 363.502,Z 378.207,A -85,B 0,C 180,E1 -13431.389,E2 -13431.389} C_VEL
LIN {X 0,Y 358.027,Z 348.939,A -85,B 0,C 180,E1 -13432.349,E2 -13432.349} C_VEL
LIN {X 0,Y 356.804,Z 343.114,A -85,B 0,C 180,E1 -13432.59,E2 -13432.59} C_VEL
LIN {X 0,Y 356.983,Z 340.899,A -85,B 0,C 180,E1 -13433.187,E2 -13433.187} C_VEL
LIN {X 0,Y 358.069,Z 331.129,A -85,B 0,C 180,E1 -13436.206,E2 -13436.206} C_VEL
LIN {X 0,Y 356.734,Z 323.046,A -85,B 0,C 180,E1 -13438.859,E2 -13438.859} C_VEL
LIN {X 0,Y 354.86,Z 313.828,A -85,B 0,C 180,E1 -13442.021,E2 -13442.021} C_VEL
LIN {X 0,Y 354.821,Z 313.773,A -85,B 0,C 180,E1 -13445.698,E2 -13445.698} C_VEL
LIN {X 0,Y 354.767,Z 313.778,A -85,B 0,C 180,E1 -13449.411,E2 -13449.411} C_VEL
LIN {X 0,Y 354.784,Z 313.79,A -85,B 0,C 180,E1 -13452.866,E2 -13452.866} C_VEL
LIN {X 0,Y 354.764,Z 313.789,A -85,B 0,C 180,E1 -13456.102,E2 -13456.102} C_VEL
LIN {X 0,Y 354.784,Z 313.786,A -85,B 0,C 180,E1 -13459.178,E2 -13459.178} C_VEL
LIN {X 0,Y 354.802,Z 313.788,A -85,B 0,C 180,E1 -13462.402,E2 -13462.402} C_VEL
LIN {X 0,Y 354.804,Z 313.779,A -85,B 0,C 180,E1 -13464.939,E2 -13464.939} C_VEL
LIN {X 0,Y 354.788,Z 313.789,A -85,B 0,C 180,E1 -13468.404,E2 -13468.404} C_VEL
LIN {X 0,Y 354.841,Z 313.771,A -85,B 0,C 180,E1 -13471.618,E2 -13471.618} C_VEL
LIN {X 0,Y 354.892,Z 313.761,A -85,B 0,C 180,E1 -13474.171,E2 -13474.171} C_VEL
LIN {X 0,Y 354.809,Z 313.784,A -85,B 0,C 180,E1 -13477.892,E2 -13477.892} C_VEL
LIN {X 0,Y 354.916,Z 313.749,A -85,B 0,C 180,E1 -13481.891,E2 -13481.891} C_VEL
LIN {X 0,Y 354.936,Z 313.769,A -85,B 0,C 180,E1 -13485.981,E2 -13485.981} C_VEL
LIN {X 0,Y 354.971,Z 313.737,A -85,B 0,C 180,E1 -13489.735,E2 -13489.735} C_VEL
LIN {X 0,Y 355.118,Z 313.739,A -85,B 0,C 180,E1 -13493.18,E2 -13493.18} C_VEL
LIN {X 0,Y 355.237,Z 313.723,A -85,B 0,C 180,E1 -13497.732,E2 -13497.732} C_VEL
LIN {X 0,Y 355.368,Z 313.685,A -85,B 0,C 180,E1 -13499.999,E2 -13499.999} C_VEL
LIN {X 0,Y 355.235,Z 313.72,A -85,B 0,C 180,E1 -13502.267,E2 -13502.267} C_VEL
LIN {X 0,Y 355.117,Z 313.747,A -85,B 0,C 180,E1 -13506.819,E2 -13506.819} C_VEL
LIN {X 0,Y 354.969,Z 313.736,A -85,B 0,C 180,E1 -13510.264,E2 -13510.264} C_VEL
LIN {X 0,Y 354.934,Z 313.77,A -85,B 0,C 180,E1 -13514.018,E2 -13514.018} C_VEL
LIN {X 0,Y 354.914,Z 313.757,A -85,B 0,C 180,E1 -13518.108,E2 -13518.108} C_VEL
LIN {X 0,Y 354.827,Z 313.781,A -85,B 0,C 180,E1 -13522.106,E2 -13522.106} C_VEL
LIN {X 0,Y 354.891,Z 313.767,A -85,B 0,C 180,E1 -13525.827,E2 -13525.827} C_VEL
LIN {X 0,Y 354.846,Z 313.78,A -85,B 0,C 180,E1 -13529.678,E2 -13529.678} C_VEL
LIN {X 0,Y 354.798,Z 313.777,A -85,B 0,C 180,E1 -13533.702,E2 -13533.702} C_VEL
LIN {X 0,Y 354.791,Z 313.786,A -85,B 0,C 180,E1 -13536.459,E2 -13536.459} C_VEL
LIN {X 0,Y 354.816,Z 313.78,A -85,B 0,C 180,E1 -13539.424,E2 -13539.424} C_VEL
LIN {X 0,Y 354.827,Z 313.788,A -85,B 0,C 180,E1 -13542.875,E2 -13542.875} C_VEL
LIN {X 0,Y 354.777,Z 313.767,A -85,B 0,C 180,E1 -13546.106,E2 -13546.106} C_VEL
LIN {X 0,Y 354.812,Z 313.754,A -85,B 0,C 180,E1 -13549.184,E2 -13549.184} C_VEL
LIN {X 0,Y 354.806,Z 313.791,A -85,B 0,C 180,E1 -13552.402,E2 -13552.402} C_VEL
LIN {X 0,Y 354.805,Z 313.76,A -85,B 0,C 180,E1 -13554.941,E2 -13554.941} C_VEL
LIN {X 0,Y 354.787,Z 313.794,A -85,B 0,C 180,E1 -13558.405,E2 -13558.405} C_VEL
LIN {X 0,Y 354.841,Z 313.771,A -85,B 0,C 180,E1 -13561.619,E2 -13561.619} C_VEL
LIN {X 0,Y 354.894,Z 313.78,A -85,B 0,C 180,E1 -13564.173,E2 -13564.173} C_VEL
LIN {X 0,Y 354.83,Z 313.788,A -85,B 0,C 180,E1 -13567.894,E2 -13567.894} C_VEL
LIN {X 0,Y 354.912,Z 314.031,A -85,B 0,C 180,E1 -13570.667,E2 -13570.667} C_VEL
LIN {X 0,Y 355.229,Z 315.271,A -85,B 0,C 180,E1 -13570.97,E2 -13570.97} C_VEL
LIN {X 0,Y 356.8,Z 317.814,A -85,B 0,C 180,E1 -13571.427,E2 -13571.427} C_VEL
LIN {X 0,Y 359.107,Z 319.69,A -85,B 0,C 180,E1 -13572.018,E2 -13572.018} C_VEL
LIN {X 0,Y 361.198,Z 322.962,A -85,B 0,C 180,E1 -13572.647,E2 -13572.647} C_VEL
LIN {X 0,Y 364.119,Z 325.44,A -85,B 0,C 180,E1 -13573.452,E2 -13573.452} C_VEL
LIN {X 0,Y 366.535,Z 328.731,A -85,B 0,C 180,E1 -13574.233,E2 -13574.233} C_VEL
LIN {X 0,Y 369.915,Z 331.494,A -85,B 0,C 180,E1 -13575.295,E2 -13575.295} C_VEL
LIN {X 0,Y 372.567,Z 334.824,A -85,B 0,C 180,E1 -13576.22,E2 -13576.22} C_VEL
LIN {X 0,Y 375.688,Z 337.213,A -85,B 0,C 180,E1 -13577.371,E2 -13577.371} C_VEL
LIN {X 0,Y 379.015,Z 341.125,A -85,B 0,C 180,E1 -13578.785,E2 -13578.785} C_VEL
LIN {X 0,Y 381.759,Z 343.24,A -85,B 0,C 180,E1 -13580.043,E2 -13580.043} C_VEL
LIN {X 0,Y 383.693,Z 344.298,A -85,B 0,C 180,E1 -13580.976,E2 -13580.976} C_VEL
LIN {X 0,Y 386.239,Z 347.585,A -85,B 0,C 180,E1 -13582.578,E2 -13582.578} C_VEL
LIN {X 0,Y 388.48,Z 349.393,A -85,B 0,C 180,E1 -13584.264,E2 -13584.264} C_VEL
LIN {X 0,Y 390.135,Z 350.327,A -85,B 0,C 180,E1 -13585.868,E2 -13585.868} C_VEL
LIN {X 0,Y 391.261,Z 350.711,A -85,B 0,C 180,E1 -13587.445,E2 -13587.445} C_VEL
LIN {X 0,Y 391.823,Z 351.132,A -85,B 0,C 180,E1 -13588.972,E2 -13588.972} C_VEL
LIN {X 0,Y 391.999,Z 351.069,A -85,B 0,C 180,E1 -13590,E2 -13590} C_VEL
LIN {X 0,Y 391.73,Z 351.018,A -85,B 0,C 180,E1 -13591.542,E2 -13591.542} C_VEL
LIN {X 0,Y 390.988,Z 350.588,A -85,B 0,C 180,E1 -13593.091,E2 -13593.091} C_VEL
LIN {X 0,Y 389.394,Z 349.977,A -85,B 0,C 180,E1 -13594.918,E2 -13594.918} C_VEL
LIN {X 0,Y 387.3,Z 348.538,A -85,B 0,C 180,E1 -13596.652,E2 -13596.652} C_VEL
LIN {X 0,Y 385.37,Z 346.629,A -85,B 0,C 180,E1 -13597.981,E2 -13597.981} C_VEL
LIN {X 0,Y 383.438,Z 344.009,A -85,B 0,C 180,E1 -13599.167,E2 -13599.167} C_VEL
LIN {X 0,Y 380.179,Z 342.115,A -85,B 0,C 180,E1 -13600.72,E2 -13600.72} C_VEL
LIN {X 0,Y 376.999,Z 338.844,A -85,B 0,C 180,E1 -13602.106,E2 -13602.106} C_VEL
LIN {X 0,Y 375.689,Z 337.211,A -85,B 0,C 180,E1 -13602.629,E2 -13602.629} C_VEL
LIN {X 0,Y 372.562,Z 334.806,A -85,B 0,C 180,E1 -13603.783,E2 -13603.783} C_VEL
LIN {X 0,Y 369.83,Z 331.406,A -85,B 0,C 180,E1 -13604.735,E2 -13604.735} C_VEL
LIN {X 0,Y 366.228,Z 328.403,A -85,B 0,C 180,E1 -13605.861,E2 -13605.861} C_VEL
LIN {X 0,Y 364.014,Z 325.235,A -85,B 0,C 180,E1 -13606.584,E2 -13606.584} C_VEL
LIN {X 0,Y 360.826,Z 322.548,A -85,B 0,C 180,E1 -13607.457,E2 -13607.457} C_VEL
LIN {X 0,Y 358.715,Z 319.221,A -85,B 0,C 180,E1 -13608.097,E2 -13608.097} C_VEL
LIN {X 0,Y 356.497,Z 317.493,A -85,B 0,C 180,E1 -13608.649,E2 -13608.649} C_VEL
LIN {X 0,Y 355.027,Z 314.607,A -85,B 0,C 180,E1 -13609.139,E2 -13609.139} C_VEL
LIN {X 0,Y 354.86,Z 313.836,A -85,B 0,C 180,E1 -13609.524,E2 -13609.524} C_VEL
LIN {X 0,Y 354.827,Z 313.789,A -85,B 0,C 180,E1 -13613.336,E2 -13613.336} C_VEL
LIN {X 0,Y 354.882,Z 313.781,A -85,B 0,C 180,E1 -13616.981,E2 -13616.981} C_VEL
LIN {X 0,Y 354.812,Z 313.77,A -85,B 0,C 180,E1 -13619.682,E2 -13619.682} C_VEL
LIN {X 0,Y 354.808,Z 313.765,A -85,B 0,C 180,E1 -13623.684,E2 -13623.684} C_VEL
LIN {X 0,Y 354.795,Z 313.782,A -85,B 0,C 180,E1 -13626.459,E2 -13626.459} C_VEL
LIN {X 0,Y 354.817,Z 313.777,A -85,B 0,C 180,E1 -13629.423,E2 -13629.423} C_VEL
LIN {X 0,Y 354.786,Z 313.752,A -85,B 0,C 180,E1 -13632.868,E2 -13632.868} C_VEL
LIN {X 0,Y 354.833,Z 313.784,A -85,B 0,C 180,E1 -13636.115,E2 -13636.115} C_VEL
LIN {X 0,Y 354.817,Z 313.774,A -85,B 0,C 180,E1 -13639.6,E2 -13639.6} C_VEL
LIN {X 0,Y 354.791,Z 313.786,A -85,B 0,C 180,E1 -13643.541,E2 -13643.541} C_VEL
LIN {X 0,Y 354.805,Z 313.778,A -85,B 0,C 180,E1 -13644.534,E2 -13644.534} C_VEL
LIN {X 0,Y 354.116,Z 313.86,A -85,B 0,C 180,E1 -13645.482,E2 -13645.482} C_VEL
LIN {X 0,Y 351.221,Z 314.227,A -85,B 0,C 180,E1 -13647.021,E2 -13647.021} C_VEL
LIN {X 0,Y 348.805,Z 314.535,A -85,B 0,C 180,E1 -13648.267,E2 -13648.267} C_VEL
LIN {X 0,Y 347.809,Z 314.662,A -85,B 0,C 180,E1 -13649.232,E2 -13649.232} C_VEL
LIN {X 0,Y 347.749,Z 314.665,A -85,B 0,C 180,E1 -13649.559,E2 -13649.559} C_VEL
LIN {X 0,Y 347.844,Z 314.633,A -85,B 0,C 180,E1 -13652.745,E2 -13652.745} C_VEL
LIN {X 0,Y 347.78,Z 314.662,A -85,B 0,C 180,E1 -13656.162,E2 -13656.162} C_VEL
LIN {X 0,Y 347.806,Z 314.639,A -85,B 0,C 180,E1 -13659.91,E2 -13659.91} C_VEL
LIN {X 0,Y 347.858,Z 314.637,A -85,B 0,C 180,E1 -13662.36,E2 -13662.36} C_VEL
LIN {X 0,Y 347.889,Z 314.648,A -85,B 0,C 180,E1 -13665.971,E2 -13665.971} C_VEL
LIN {X 0,Y 347.92,Z 314.614,A -85,B 0,C 180,E1 -13669.526,E2 -13669.526} C_VEL
LIN {X 0,Y 348.083,Z 314.621,A -85,B 0,C 180,E1 -13673.043,E2 -13673.043} C_VEL
LIN {X 0,Y 348.198,Z 314.597,A -85,B 0,C 180,E1 -13677.687,E2 -13677.687} C_VEL
LIN {X 0,Y 348.318,Z 314.562,A -85,B 0,C 180,E1 -13680.001,E2 -13680.001} C_VEL
LIN {X 0,Y 348.2,Z 314.6,A -85,B 0,C 180,E1 -13682.314,E2 -13682.314} C_VEL
LIN {X 0,Y 348.084,Z 314.614,A -85,B 0,C 180,E1 -13686.959,E2 -13686.959} C_VEL
LIN {X 0,Y 347.921,Z 314.617,A -85,B 0,C 180,E1 -13690.475,E2 -13690.475} C_VEL
LIN {X 0,Y 347.892,Z 314.647,A -85,B 0,C 180,E1 -13694.151,E2 -13694.151} C_VEL
LIN {X 0,Y 347.885,Z 314.623,A -85,B 0,C 180,E1 -13698.291,E2 -13698.291} C_VEL
LIN {X 0,Y 347.761,Z 314.66,A -85,B 0,C 180,E1 -13701.627,E2 -13701.627} C_VEL
LIN {X 0,Y 347.805,Z 314.648,A -85,B 0,C 180,E1 -13705.11,E2 -13705.11} C_VEL
LIN {X 0,Y 347.803,Z 314.642,A -85,B 0,C 180,E1 -13707.695,E2 -13707.695} C_VEL
LIN {X 0,Y 347.744,Z 314.67,A -85,B 0,C 180,E1 -13710.349,E2 -13710.349} C_VEL
LIN {X 0,Y 347.744,Z 314.651,A -85,B 0,C 180,E1 -13714.045,E2 -13714.045} C_VEL
LIN {X 0,Y 347.756,Z 314.665,A -85,B 0,C 180,E1 -13717.322,E2 -13717.322} C_VEL
LIN {X 0,Y 347.729,Z 314.66,A -85,B 0,C 180,E1 -13720.298,E2 -13720.298} C_VEL
LIN {X 0,Y 347.721,Z 314.669,A -85,B 0,C 180,E1 -13723.409,E2 -13723.409} C_VEL
LIN {X 0,Y 347.723,Z 314.671,A -85,B 0,C 180,E1 -13726.688,E2 -13726.688} C_VEL
LIN {X 0,Y 347.7,Z 314.653,A -85,B 0,C 180,E1 -13730.183,E2 -13730.183} C_VEL
LIN {X 0,Y 347.756,Z 314.665,A -85,B 0,C 180,E1 -13732.68,E2 -13732.68} C_VEL
LIN {X 0,Y 347.748,Z 314.67,A -85,B 0,C 180,E1 -13735.957,E2 -13735.957} C_VEL
LIN {X 0,Y 347.817,Z 314.881,A -85,B 0,C 180,E1 -13737.704,E2 -13737.704} C_VEL
LIN {X 0,Y 349.433,Z 322.823,A -85,B 0,C 180,E1 -13740.571,E2 -13740.571} C_VEL
LIN {X 0,Y 350.938,Z 330.904,A -85,B 0,C 180,E1 -13743.219,E2 -13743.219} C_VEL
LIN {X 0,Y 350.992,Z 334.257,A -85,B 0,C 180,E1 -13744.297,E2 -13744.297} C_VEL
LIN {X 0,Y 349.962,Z 342.719,A -85,B 0,C 180,E1 -13746.913,E2 -13746.913} C_VEL
LIN {X 0,Y 350.755,Z 346.818,A -85,B 0,C 180,E1 -13747.12,E2 -13747.12} C_VEL
LIN {X 0,Y 356.254,Z 375.353,A -85,B 0,C 180,E1 -13748.097,E2 -13748.097} C_VEL
LIN {X 0,Y 356.918,Z 381.27,A -85,B 0,C 180,E1 -13748.265,E2 -13748.265} C_VEL
LIN {X 0,Y 355.693,Z 447.654,A -85,B 0,C 180,E1 -13749.62,E2 -13749.62} C_VEL
LIN {X 0,Y 355.216,Z 458.411,A -85,B 0,C 180,E1 -13749.969,E2 -13749.969} C_VEL
LIN {X 0,Y 354.605,Z 467.508,A -85,B 0,C 180,E1 -13750.386,E2 -13750.386} C_VEL
LIN {X 0,Y 353.839,Z 476.861,A -85,B 0,C 180,E1 -13750.945,E2 -13750.945} C_VEL
LIN {X 0,Y 352.9,Z 487,A -85,B 0,C 180,E1 -13751.72,E2 -13751.72} C_VEL
LIN {X 0,Y 351.928,Z 495.994,A -85,B 0,C 180,E1 -13752.57,E2 -13752.57} C_VEL
LIN {X 0,Y 350.948,Z 504.721,A -85,B 0,C 180,E1 -13753.569,E2 -13753.569} C_VEL
LIN {X 0,Y 350.067,Z 512.82,A -85,B 0,C 180,E1 -13754.683,E2 -13754.683} C_VEL
LIN {X 0,Y 349.089,Z 520.964,A -85,B 0,C 180,E1 -13756.02,E2 -13756.02} C_VEL
LIN {X 0,Y 348.371,Z 526.915,A -85,B 0,C 180,E1 -13757.179,E2 -13757.179} C_VEL
LIN {X 0,Y 347.567,Z 533.23,A -85,B 0,C 180,E1 -13758.63,E2 -13758.63} C_VEL
LIN {X 0,Y 347.022,Z 538.493,A -85,B 0,C 180,E1 -13760.088,E2 -13760.088} C_VEL
LIN {X 0,Y 346.56,Z 543.624,A -85,B 0,C 180,E1 -13761.839,E2 -13761.839} C_VEL
LIN {X 0,Y 346.284,Z 547.614,A -85,B 0,C 180,E1 -13763.592,E2 -13763.592} C_VEL
LIN {X 0,Y 346.162,Z 550.563,A -85,B 0,C 180,E1 -13765.342,E2 -13765.342} C_VEL
LIN {X 0,Y 346.084,Z 553.008,A -85,B 0,C 180,E1 -13767.672,E2 -13767.672} C_VEL
LIN {X 0,Y 346.104,Z 553.597,A -85,B 0,C 180,E1 -13768.836,E2 -13768.836} C_VEL
LIN {X 0,Y 346.104,Z 553.597,A -85,B 0,C 180,E1 -13771.164,E2 -13771.164} C_VEL
LIN {X 0,Y 346.084,Z 553.008,A -85,B 0,C 180,E1 -13772.328,E2 -13772.328} C_VEL
LIN {X 0,Y 346.161,Z 550.563,A -85,B 0,C 180,E1 -13774.658,E2 -13774.658} C_VEL
LIN {X 0,Y 346.247,Z 547.613,A -85,B 0,C 180,E1 -13776.409,E2 -13776.409} C_VEL
LIN {X 0,Y 346.56,Z 543.624,A -85,B 0,C 180,E1 -13778.161,E2 -13778.161} C_VEL
LIN {X 0,Y 347.022,Z 538.493,A -85,B 0,C 180,E1 -13779.912,E2 -13779.912} C_VEL
LIN {X 0,Y 347.567,Z 533.23,A -85,B 0,C 180,E1 -13781.37,E2 -13781.37} C_VEL
LIN {X 0,Y 348.357,Z 526.915,A -85,B 0,C 180,E1 -13782.822,E2 -13782.822} C_VEL
LIN {X 0,Y 349.114,Z 520.965,A -85,B 0,C 180,E1 -13783.979,E2 -13783.979} C_VEL
LIN {X 0,Y 350.042,Z 512.925,A -85,B 0,C 180,E1 -13785.302,E2 -13785.302} C_VEL
LIN {X 0,Y 350.965,Z 504.721,A -85,B 0,C 180,E1 -13786.43,E2 -13786.43} C_VEL
LIN {X 0,Y 351.955,Z 495.995,A -85,B 0,C 180,E1 -13787.429,E2 -13787.429} C_VEL
LIN {X 0,Y 352.906,Z 487,A -85,B 0,C 180,E1 -13788.279,E2 -13788.279} C_VEL
LIN {X 0,Y 353.822,Z 476.86,A -85,B 0,C 180,E1 -13789.056,E2 -13789.056} C_VEL
LIN {X 0,Y 354.796,Z 464.933,A -85,B 0,C 180,E1 -13789.754,E2 -13789.754} C_VEL
LIN {X 0,Y 355.547,Z 451.64,A -85,B 0,C 180,E1 -13790.275,E2 -13790.275} C_VEL
LIN {X 0,Y 356.003,Z 432.862,A -85,B 0,C 180,E1 -13790.701,E2 -13790.701} C_VEL
LIN {X 0,Y 356.823,Z 378.718,A -85,B 0,C 180,E1 -13791.795,E2 -13791.795} C_VEL
LIN {X 0,Y 351.518,Z 350.422,A -85,B 0,C 180,E1 -13792.75,E2 -13792.75} C_VEL
LIN {X 0,Y 349.951,Z 342.994,A -85,B 0,C 180,E1 -13793.05,E2 -13793.05} C_VEL
LIN {X 0,Y 350.017,Z 341.647,A -85,B 0,C 180,E1 -13793.363,E2 -13793.363} C_VEL
LIN {X 0,Y 351.071,Z 332.925,A -85,B 0,C 180,E1 -13796.13,E2 -13796.13} C_VEL
LIN {X 0,Y 350.153,Z 326.278,A -85,B 0,C 180,E1 -13798.341,E2 -13798.341} C_VEL
LIN {X 0,Y 348.208,Z 316.604,A -85,B 0,C 180,E1 -13801.652,E2 -13801.652} C_VEL
LIN {X 0,Y 347.781,Z 314.677,A -85,B 0,C 180,E1 -13802.452,E2 -13802.452} C_VEL
LIN {X 0,Y 347.769,Z 314.651,A -85,B 0,C 180,E1 -13806.064,E2 -13806.064} C_VEL
LIN {X 0,Y 347.73,Z 314.666,A -85,B 0,C 180,E1 -13808.794,E2 -13808.794} C_VEL
LIN {X 0,Y 347.742,Z 314.653,A -85,B 0,C 180,E1 -13811.83,E2 -13811.83} C_VEL
LIN {X 0,Y 347.703,Z 314.669,A -85,B 0,C 180,E1 -13815.026,E2 -13815.026} C_VEL
LIN {X 0,Y 347.747,Z 314.665,A -85,B 0,C 180,E1 -13818.396,E2 -13818.396} C_VEL
LIN {X 0,Y 347.769,Z 314.666,A -85,B 0,C 180,E1 -13822.011,E2 -13822.011} C_VEL
LIN {X 0,Y 347.739,Z 314.653,A -85,B 0,C 180,E1 -13825.535,E2 -13825.535} C_VEL
LIN {X 0,Y 347.74,Z 314.667,A -85,B 0,C 180,E1 -13828.299,E2 -13828.299} C_VEL
LIN {X 0,Y 347.774,Z 314.661,A -85,B 0,C 180,E1 -13830.987,E2 -13830.987} C_VEL
LIN {X 0,Y 347.825,Z 314.636,A -85,B 0,C 180,E1 -13833.607,E2 -13833.607} C_VEL
LIN {X 0,Y 347.779,Z 314.661,A -85,B 0,C 180,E1 -13836.161,E2 -13836.161} C_VEL
LIN {X 0,Y 347.8,Z 314.642,A -85,B 0,C 180,E1 -13839.908,E2 -13839.908} C_VEL
LIN {X 0,Y 347.86,Z 314.631,A -85,B 0,C 180,E1 -13842.358,E2 -13842.358} C_VEL
LIN {X 0,Y 347.891,Z 314.647,A -85,B 0,C 180,E1 -13845.97,E2 -13845.97} C_VEL
LIN {X 0,Y 347.921,Z 314.617,A -85,B 0,C 180,E1 -13849.525,E2 -13849.525} C_VEL
LIN {X 0,Y 348.084,Z 314.614,A -85,B 0,C 180,E1 -13853.041,E2 -13853.041} C_VEL
LIN {X 0,Y 348.2,Z 314.6,A -85,B 0,C 180,E1 -13857.686,E2 -13857.686} C_VEL
LIN {X 0,Y 348.318,Z 314.562,A -85,B 0,C 180,E1 -13859.999,E2 -13859.999} C_VEL
LIN {X 0,Y 348.198,Z 314.597,A -85,B 0,C 180,E1 -13862.313,E2 -13862.313} C_VEL
LIN {X 0,Y 348.083,Z 314.621,A -85,B 0,C 180,E1 -13866.957,E2 -13866.957} C_VEL
LIN {X 0,Y 347.92,Z 314.614,A -85,B 0,C 180,E1 -13870.474,E2 -13870.474} C_VEL
LIN {X 0,Y 347.89,Z 314.648,A -85,B 0,C 180,E1 -13874.149,E2 -13874.149} C_VEL
LIN {X 0,Y 347.882,Z 314.63,A -85,B 0,C 180,E1 -13878.29,E2 -13878.29} C_VEL
LIN {X 0,Y 347.781,Z 314.659,A -85,B 0,C 180,E1 -13881.635,E2 -13881.635} C_VEL
LIN {X 0,Y 347.803,Z 314.654,A -85,B 0,C 180,E1 -13885.108,E2 -13885.108} C_VEL
LIN {X 0,Y 347.804,Z 314.639,A -85,B 0,C 180,E1 -13887.694,E2 -13887.694} C_VEL
LIN {X 0,Y 347.757,Z 314.665,A -85,B 0,C 180,E1 -13890.346,E2 -13890.346} C_VEL
LIN {X 0,Y 347.736,Z 314.653,A -85,B 0,C 180,E1 -13894.464,E2 -13894.464} C_VEL
LIN {X 0,Y 347.768,Z 314.665,A -85,B 0,C 180,E1 -13897.989,E2 -13897.989} C_VEL
LIN {X 0,Y 347.776,Z 314.657,A -85,B 0,C 180,E1 -13901.609,E2 -13901.609} C_VEL
LIN {X 0,Y 347.79,Z 314.653,A -85,B 0,C 180,E1 -13905.012,E2 -13905.012} C_VEL
LIN {X 0,Y 347.755,Z 314.623,A -85,B 0,C 180,E1 -13908.395,E2 -13908.395} C_VEL
LIN {X 0,Y 347.771,Z 314.666,A -85,B 0,C 180,E1 -13912.011,E2 -13912.011} C_VEL
LIN {X 0,Y 347.738,Z 314.639,A -85,B 0,C 180,E1 -13915.536,E2 -13915.536} C_VEL
LIN {X 0,Y 347.739,Z 314.672,A -85,B 0,C 180,E1 -13918.301,E2 -13918.301} C_VEL
LIN {X 0,Y 347.773,Z 314.646,A -85,B 0,C 180,E1 -13920.988,E2 -13920.988} C_VEL
LIN {X 0,Y 347.826,Z 314.66,A -85,B 0,C 180,E1 -13923.608,E2 -13923.608} C_VEL
LIN {X 0,Y 347.784,Z 314.666,A -85,B 0,C 180,E1 -13926.162,E2 -13926.162} C_VEL
LIN {X 0,Y 347.82,Z 314.783,A -85,B 0,C 180,E1 -13929.138,E2 -13929.138} C_VEL
LIN {X 0,Y 348.019,Z 315.803,A -85,B 0,C 180,E1 -13929.459,E2 -13929.459} C_VEL
LIN {X 0,Y 349.599,Z 318.571,A -85,B 0,C 180,E1 -13929.907,E2 -13929.907} C_VEL
LIN {X 0,Y 351.929,Z 320.639,A -85,B 0,C 180,E1 -13930.441,E2 -13930.441} C_VEL
LIN {X 0,Y 353.933,Z 323.736,A -85,B 0,C 180,E1 -13930.994,E2 -13930.994} C_VEL
LIN {X 0,Y 356.537,Z 326.105,A -85,B 0,C 180,E1 -13931.643,E2 -13931.643} C_VEL
LIN {X 0,Y 358.935,Z 329.401,A -85,B 0,C 180,E1 -13932.324,E2 -13932.324} C_VEL
LIN {X 0,Y 361.877,Z 332.028,A -85,B 0,C 180,E1 -13933.127,E2 -13933.127} C_VEL
LIN {X 0,Y 364.75,Z 335.483,A -85,B 0,C 180,E1 -13934.011,E2 -13934.011} C_VEL
LIN {X 0,Y 367.928,Z 338.098,A -85,B 0,C 180,E1 -13934.968,E2 -13934.968} C_VEL
LIN {X 0,Y 370.999,Z 341.699,A -85,B 0,C 180,E1 -13936.035,E2 -13936.035} C_VEL
LIN {X 0,Y 374.676,Z 344.691,A -85,B 0,C 180,E1 -13937.369,E2 -13937.369} C_VEL
LIN {X 0,Y 377.469,Z 347.844,A -85,B 0,C 180,E1 -13938.533,E2 -13938.533} C_VEL
LIN {X 0,Y 380.55,Z 350.172,A -85,B 0,C 180,E1 -13939.902,E2 -13939.902} C_VEL
LIN {X 0,Y 382.425,Z 351.252,A -85,B 0,C 180,E1 -13940.794,E2 -13940.794} C_VEL
LIN {X 0,Y 385.152,Z 354.564,A -85,B 0,C 180,E1 -13942.453,E2 -13942.453} C_VEL
LIN {X 0,Y 387.586,Z 356.461,A -85,B 0,C 180,E1 -13944.251,E2 -13944.251} C_VEL
LIN {X 0,Y 389.26,Z 357.372,A -85,B 0,C 180,E1 -13945.859,E2 -13945.859} C_VEL
LIN {X 0,Y 390.395,Z 357.749,A -85,B 0,C 180,E1 -13947.439,E2 -13947.439} C_VEL
LIN {X 0,Y 390.961,Z 358.179,A -85,B 0,C 180,E1 -13948.97,E2 -13948.97} C_VEL
LIN {X 0,Y 391.134,Z 358.116,A -85,B 0,C 180,E1 -13950,E2 -13950} C_VEL
LIN {X 0,Y 390.861,Z 358.065,A -85,B 0,C 180,E1 -13951.545,E2 -13951.545} C_VEL
LIN {X 0,Y 390.115,Z 357.609,A -85,B 0,C 180,E1 -13953.098,E2 -13953.098} C_VEL
LIN {X 0,Y 388.503,Z 357.03,A -85,B 0,C 180,E1 -13954.929,E2 -13954.929} C_VEL
LIN {X 0,Y 386.387,Z 355.616,A -85,B 0,C 180,E1 -13956.668,E2 -13956.668} C_VEL
LIN {X 0,Y 384.294,Z 353.698,A -85,B 0,C 180,E1 -13958.072,E2 -13958.072} C_VEL
LIN {X 0,Y 382.055,Z 350.873,A -85,B 0,C 180,E1 -13959.396,E2 -13959.396} C_VEL
LIN {X 0,Y 378.834,Z 348.992,A -85,B 0,C 180,E1 -13960.894,E2 -13960.894} C_VEL
LIN {X 0,Y 375.554,Z 345.766,A -85,B 0,C 180,E1 -13962.29,E2 -13962.29} C_VEL
LIN {X 0,Y 373.857,Z 343.853,A -85,B 0,C 180,E1 -13962.942,E2 -13962.942} C_VEL
LIN {X 0,Y 370.854,Z 341.557,A -85,B 0,C 180,E1 -13964.014,E2 -13964.014} C_VEL
LIN {X 0,Y 367.856,Z 337.994,A -85,B 0,C 180,E1 -13965.057,E2 -13965.057} C_VEL
LIN {X 0,Y 363.527,Z 334.208,A -85,B 0,C 180,E1 -13966.37,E2 -13966.37} C_VEL
LIN {X 0,Y 361.121,Z 331.195,A -85,B 0,C 180,E1 -13967.082,E2 -13967.082} C_VEL
LIN {X 0,Y 358.257,Z 328.628,A -85,B 0,C 180,E1 -13967.871,E2 -13967.871} C_VEL
LIN {X 0,Y 356.112,Z 325.524,A -85,B 0,C 180,E1 -13968.468,E2 -13968.468} C_VEL
LIN {X 0,Y 353.384,Z 323.096,A -85,B 0,C 180,E1 -13969.15,E2 -13969.15} C_VEL
LIN {X 0,Y 351.55,Z 320.073,A -85,B 0,C 180,E1 -13969.658,E2 -13969.658} C_VEL
LIN {X 0,Y 349.253,Z 318.187,A -85,B 0,C 180,E1 -13970.175,E2 -13970.175} C_VEL
LIN {X 0,Y 347.917,Z 315.338,A -85,B 0,C 180,E1 -13970.624,E2 -13970.624} C_VEL
LIN {X 0,Y 347.811,Z 314.699,A -85,B 0,C 180,E1 -13971.018,E2 -13971.018} C_VEL
LIN {X 0,Y 347.807,Z 314.663,A -85,B 0,C 180,E1 -13975.108,E2 -13975.108} C_VEL
LIN {X 0,Y 347.803,Z 314.658,A -85,B 0,C 180,E1 -13977.694,E2 -13977.694} C_VEL
LIN {X 0,Y 347.743,Z 314.656,A -85,B 0,C 180,E1 -13980.348,E2 -13980.348} C_VEL
LIN {X 0,Y 347.742,Z 314.641,A -85,B 0,C 180,E1 -13984.044,E2 -13984.044} C_VEL
LIN {X 0,Y 347.76,Z 314.665,A -85,B 0,C 180,E1 -13987.32,E2 -13987.32} C_VEL
LIN {X 0,Y 347.745,Z 314.643,A -85,B 0,C 180,E1 -13990.294,E2 -13990.294} C_VEL
LIN {X 0,Y 347.722,Z 314.637,A -85,B 0,C 180,E1 -13993.407,E2 -13993.407} C_VEL
LIN {X 0,Y 347.776,Z 314.664,A -85,B 0,C 180,E1 -13996.676,E2 -13996.676} C_VEL
LIN {X 0,Y 347.778,Z 314.656,A -85,B 0,C 180,E1 -14000.165,E2 -14000.165} C_VEL
LIN {X 0,Y 347.781,Z 314.655,A -85,B 0,C 180,E1 -14004.125,E2 -14004.125} C_VEL
LIN {X 0,Y 347.733,Z 314.668,A -85,B 0,C 180,E1 -14008.086,E2 -14008.086} C_VEL
LIN {X 0,Y 347.749,Z 314.665,A -85,B 0,C 180,E1 -14009.559,E2 -14009.559} C_VEL
LIN {X 0,Y 347.142,Z 314.744,A -85,B 0,C 180,E1 -14010.526,E2 -14010.526} C_VEL
LIN {X 0,Y 344.317,Z 315.09,A -85,B 0,C 180,E1 -14012.101,E2 -14012.101} C_VEL
LIN {X 0,Y 341.887,Z 315.387,A -85,B 0,C 180,E1 -14013.376,E2 -14013.376} C_VEL
LIN {X 0,Y 340.839,Z 315.518,A -85,B 0,C 180,E1 -14014.362,E2 -14014.362} C_VEL
LIN {X 0,Y 340.753,Z 315.53,A -85,B 0,C 180,E1 -14014.697,E2 -14014.697} C_VEL
LIN {X 0,Y 340.733,Z 315.536,A -85,B 0,C 180,E1 -14018.207,E2 -14018.207} C_VEL
LIN {X 0,Y 340.849,Z 315.508,A -85,B 0,C 180,E1 -14021.985,E2 -14021.985} C_VEL
LIN {X 0,Y 340.861,Z 315.524,A -85,B 0,C 180,E1 -14025.705,E2 -14025.705} C_VEL
LIN {X 0,Y 340.862,Z 315.493,A -85,B 0,C 180,E1 -14029.307,E2 -14029.307} C_VEL
LIN {X 0,Y 341.051,Z 315.494,A -85,B 0,C 180,E1 -14032.898,E2 -14032.898} C_VEL
LIN {X 0,Y 341.16,Z 315.473,A -85,B 0,C 180,E1 -14037.639,E2 -14037.639} C_VEL
LIN {X 0,Y 341.269,Z 315.439,A -85,B 0,C 180,E1 -14040.001,E2 -14040.001} C_VEL
LIN {X 0,Y 341.162,Z 315.477,A -85,B 0,C 180,E1 -14042.362,E2 -14042.362} C_VEL
LIN {X 0,Y 341.052,Z 315.488,A -85,B 0,C 180,E1 -14047.103,E2 -14047.103} C_VEL
LIN {X 0,Y 340.864,Z 315.498,A -85,B 0,C 180,E1 -14050.695,E2 -14050.695} C_VEL
LIN {X 0,Y 340.857,Z 315.525,A -85,B 0,C 180,E1 -14054.326,E2 -14054.326} C_VEL
LIN {X 0,Y 340.831,Z 315.5,A -85,B 0,C 180,E1 -14058.467,E2 -14058.467} C_VEL
LIN {X 0,Y 340.712,Z 315.538,A -85,B 0,C 180,E1 -14061.843,E2 -14061.843} C_VEL
LIN {X 0,Y 340.766,Z 315.521,A -85,B 0,C 180,E1 -14065.666,E2 -14065.666} C_VEL
LIN {X 0,Y 340.724,Z 315.528,A -85,B 0,C 180,E1 -14068.322,E2 -14068.322} C_VEL
LIN {X 0,Y 340.693,Z 315.545,A -85,B 0,C 180,E1 -14071.046,E2 -14071.046} C_VEL
LIN {X 0,Y 340.712,Z 315.535,A -85,B 0,C 180,E1 -14075.28,E2 -14075.28} C_VEL
LIN {X 0,Y 340.705,Z 315.541,A -85,B 0,C 180,E1 -14078.387,E2 -14078.387} C_VEL
LIN {X 0,Y 340.696,Z 315.547,A -85,B 0,C 180,E1 -14082.046,E2 -14082.046} C_VEL
LIN {X 0,Y 340.65,Z 315.556,A -85,B 0,C 180,E1 -14086.228,E2 -14086.228} C_VEL
LIN {X 0,Y 340.669,Z 315.528,A -85,B 0,C 180,E1 -14088.689,E2 -14088.689} C_VEL
LIN {X 0,Y 340.718,Z 315.544,A -85,B 0,C 180,E1 -14091.772,E2 -14091.772} C_VEL
LIN {X 0,Y 340.723,Z 315.54,A -85,B 0,C 180,E1 -14095.596,E2 -14095.596} C_VEL
LIN {X 0,Y 340.755,Z 315.734,A -85,B 0,C 180,E1 -14097.31,E2 -14097.31} C_VEL
LIN {X 0,Y 342.303,Z 323.198,A -85,B 0,C 180,E1 -14100.078,E2 -14100.078} C_VEL
LIN {X 0,Y 343.896,Z 331.735,A -85,B 0,C 180,E1 -14102.954,E2 -14102.954} C_VEL
LIN {X 0,Y 344.087,Z 334.805,A -85,B 0,C 180,E1 -14103.989,E2 -14103.989} C_VEL
LIN {X 0,Y 343.09,Z 342.438,A -85,B 0,C 180,E1 -14106.407,E2 -14106.407} C_VEL
LIN {X 0,Y 343.42,Z 344.395,A -85,B 0,C 180,E1 -14106.552,E2 -14106.552} C_VEL
LIN {X 0,Y 348.63,Z 370.374,A -85,B 0,C 180,E1 -14107.489,E2 -14107.489} C_VEL
LIN {X 0,Y 350.342,Z 381.076,A -85,B 0,C 180,E1 -14107.836,E2 -14107.836} C_VEL
LIN {X 0,Y 349.049,Z 447.466,A -85,B 0,C 180,E1 -14109.215,E2 -14109.215} C_VEL
LIN {X 0,Y 348.54,Z 458.217,A -85,B 0,C 180,E1 -14109.569,E2 -14109.569} C_VEL
LIN {X 0,Y 347.921,Z 467.314,A -85,B 0,C 180,E1 -14109.993,E2 -14109.993} C_VEL
LIN {X 0,Y 347.029,Z 477.673,A -85,B 0,C 180,E1 -14110.633,E2 -14110.633} C_VEL
LIN {X 0,Y 346.165,Z 486.806,A -85,B 0,C 180,E1 -14111.352,E2 -14111.352} C_VEL
LIN {X 0,Y 345.138,Z 495.799,A -85,B 0,C 180,E1 -14112.216,E2 -14112.216} C_VEL
LIN {X 0,Y 344.114,Z 504.526,A -85,B 0,C 180,E1 -14113.233,E2 -14113.233} C_VEL
LIN {X 0,Y 343.174,Z 512.768,A -85,B 0,C 180,E1 -14114.39,E2 -14114.39} C_VEL
LIN {X 0,Y 342.161,Z 520.769,A -85,B 0,C 180,E1 -14115.731,E2 -14115.731} C_VEL
LIN {X 0,Y 341.421,Z 526.72,A -85,B 0,C 180,E1 -14116.913,E2 -14116.913} C_VEL
LIN {X 0,Y 340.574,Z 533.035,A -85,B 0,C 180,E1 -14118.393,E2 -14118.393} C_VEL
LIN {X 0,Y 339.998,Z 538.299,A -85,B 0,C 180,E1 -14119.881,E2 -14119.881} C_VEL
LIN {X 0,Y 339.518,Z 543.43,A -85,B 0,C 180,E1 -14121.669,E2 -14121.669} C_VEL
LIN {X 0,Y 339.205,Z 547.418,A -85,B 0,C 180,E1 -14123.457,E2 -14123.457} C_VEL
LIN {X 0,Y 339.065,Z 550.368,A -85,B 0,C 180,E1 -14125.244,E2 -14125.244} C_VEL
LIN {X 0,Y 338.999,Z 552.814,A -85,B 0,C 180,E1 -14127.624,E2 -14127.624} C_VEL
LIN {X 0,Y 339.007,Z 553.404,A -85,B 0,C 180,E1 -14128.812,E2 -14128.812} C_VEL
LIN {X 0,Y 339.007,Z 553.404,A -85,B 0,C 180,E1 -14131.188,E2 -14131.188} C_VEL
LIN {X 0,Y 338.999,Z 552.814,A -85,B 0,C 180,E1 -14132.376,E2 -14132.376} C_VEL
LIN {X 0,Y 339.064,Z 550.368,A -85,B 0,C 180,E1 -14134.756,E2 -14134.756} C_VEL
LIN {X 0,Y 339.17,Z 547.417,A -85,B 0,C 180,E1 -14136.544,E2 -14136.544} C_VEL
LIN {X 0,Y 339.518,Z 543.43,A -85,B 0,C 180,E1 -14138.331,E2 -14138.331} C_VEL
LIN {X 0,Y 339.998,Z 538.299,A -85,B 0,C 180,E1 -14140.119,E2 -14140.119} C_VEL
LIN {X 0,Y 340.574,Z 533.035,A -85,B 0,C 180,E1 -14141.607,E2 -14141.607} C_VEL
LIN {X 0,Y 341.413,Z 526.72,A -85,B 0,C 180,E1 -14143.087,E2 -14143.087} C_VEL
LIN {X 0,Y 342.183,Z 520.769,A -85,B 0,C 180,E1 -14144.268,E2 -14144.268} C_VEL
LIN {X 0,Y 343.138,Z 512.826,A -85,B 0,C 180,E1 -14145.602,E2 -14145.602} C_VEL
LIN {X 0,Y 343.997,Z 505.661,A -85,B 0,C 180,E1 -14146.62,E2 -14146.62} C_VEL
LIN {X 0,Y 345.017,Z 497.152,A -85,B 0,C 180,E1 -14147.638,E2 -14147.638} C_VEL
LIN {X 0,Y 345.988,Z 488.437,A -85,B 0,C 180,E1 -14148.505,E2 -14148.505} C_VEL
LIN {X 0,Y 346.934,Z 478.68,A -85,B 0,C 180,E1 -14149.296,E2 -14149.296} C_VEL
LIN {X 0,Y 347.789,Z 468.601,A -85,B 0,C 180,E1 -14149.938,E2 -14149.938} C_VEL
LIN {X 0,Y 348.461,Z 459.09,A -85,B 0,C 180,E1 -14150.398,E2 -14150.398} C_VEL
LIN {X 0,Y 349.005,Z 448.784,A -85,B 0,C 180,E1 -14150.749,E2 -14150.749} C_VEL
LIN {X 0,Y 350.157,Z 390.54,A -85,B 0,C 180,E1 -14151.972,E2 -14151.972} C_VEL
LIN {X 0,Y 350.283,Z 379.827,A -85,B 0,C 180,E1 -14152.195,E2 -14152.195} C_VEL
LIN {X 0,Y 345.146,Z 352.364,A -85,B 0,C 180,E1 -14153.147,E2 -14153.147} C_VEL
LIN {X 0,Y 343.102,Z 342.729,A -85,B 0,C 180,E1 -14153.544,E2 -14153.544} C_VEL
LIN {X 0,Y 343.322,Z 340.508,A -85,B 0,C 180,E1 -14154.167,E2 -14154.167} C_VEL
LIN {X 0,Y 344.105,Z 334.02,A -85,B 0,C 180,E1 -14156.27,E2 -14156.27} C_VEL
LIN {X 0,Y 343.273,Z 328.04,A -85,B 0,C 180,E1 -14158.313,E2 -14158.313} C_VEL
LIN {X 0,Y 341.395,Z 318.637,A -85,B 0,C 180,E1 -14161.621,E2 -14161.621} C_VEL
LIN {X 0,Y 340.729,Z 315.602,A -85,B 0,C 180,E1 -14162.781,E2 -14162.781} C_VEL
LIN {X 0,Y 340.708,Z 315.532,A -85,B 0,C 180,E1 -14166.439,E2 -14166.439} C_VEL
LIN {X 0,Y 340.654,Z 315.53,A -85,B 0,C 180,E1 -14169.758,E2 -14169.758} C_VEL
LIN {X 0,Y 340.672,Z 315.548,A -85,B 0,C 180,E1 -14172.904,E2 -14172.904} C_VEL
LIN {X 0,Y 340.673,Z 315.547,A -85,B 0,C 180,E1 -14177.095,E2 -14177.095} C_VEL
LIN {X 0,Y 340.696,Z 315.535,A -85,B 0,C 180,E1 -14180.246,E2 -14180.246} C_VEL
LIN {X 0,Y 340.704,Z 315.545,A -85,B 0,C 180,E1 -14183.559,E2 -14183.559} C_VEL
LIN {X 0,Y 340.688,Z 315.529,A -85,B 0,C 180,E1 -14186.152,E2 -14186.152} C_VEL
LIN {X 0,Y 340.737,Z 315.538,A -85,B 0,C 180,E1 -14190.328,E2 -14190.328} C_VEL
LIN {X 0,Y 340.798,Z 315.51,A -85,B 0,C 180,E1 -14193.019,E2 -14193.019} C_VEL
LIN {X 0,Y 340.749,Z 315.533,A -85,B 0,C 180,E1 -14195.637,E2 -14195.637} C_VEL
LIN {X 0,Y 340.728,Z 315.527,A -85,B 0,C 180,E1 -14199.472,E2 -14199.472} C_VEL
LIN {X 0,Y 340.851,Z 315.499,A -85,B 0,C 180,E1 -14201.983,E2 -14201.983} C_VEL
LIN {X 0,Y 340.863,Z 315.524,A -85,B 0,C 180,E1 -14205.704,E2 -14205.704} C_VEL
LIN {X 0,Y 340.864,Z 315.498,A -85,B 0,C 180,E1 -14209.305,E2 -14209.305} C_VEL
LIN {X 0,Y 341.052,Z 315.488,A -85,B 0,C 180,E1 -14212.897,E2 -14212.897} C_VEL
LIN {X 0,Y 341.162,Z 315.477,A -85,B 0,C 180,E1 -14217.638,E2 -14217.638} C_VEL
LIN {X 0,Y 341.269,Z 315.439,A -85,B 0,C 180,E1 -14219.999,E2 -14219.999} C_VEL
LIN {X 0,Y 341.16,Z 315.473,A -85,B 0,C 180,E1 -14222.361,E2 -14222.361} C_VEL
LIN {X 0,Y 341.051,Z 315.494,A -85,B 0,C 180,E1 -14227.102,E2 -14227.102} C_VEL
LIN {X 0,Y 340.862,Z 315.493,A -85,B 0,C 180,E1 -14230.693,E2 -14230.693} C_VEL
LIN {X 0,Y 340.855,Z 315.524,A -85,B 0,C 180,E1 -14234.324,E2 -14234.324} C_VEL
LIN {X 0,Y 340.829,Z 315.505,A -85,B 0,C 180,E1 -14238.466,E2 -14238.466} C_VEL
LIN {X 0,Y 340.746,Z 315.535,A -85,B 0,C 180,E1 -14241.857,E2 -14241.857} C_VEL
LIN {X 0,Y 340.764,Z 315.527,A -85,B 0,C 180,E1 -14245.664,E2 -14245.664} C_VEL
LIN {X 0,Y 340.734,Z 315.522,A -85,B 0,C 180,E1 -14248.319,E2 -14248.319} C_VEL
LIN {X 0,Y 340.697,Z 315.548,A -85,B 0,C 180,E1 -14251.044,E2 -14251.044} C_VEL
LIN {X 0,Y 340.71,Z 315.531,A -85,B 0,C 180,E1 -14255.279,E2 -14255.279} C_VEL
LIN {X 0,Y 340.711,Z 315.547,A -85,B 0,C 180,E1 -14258.388,E2 -14258.388} C_VEL
LIN {X 0,Y 340.717,Z 315.533,A -85,B 0,C 180,E1 -14261.304,E2 -14261.304} C_VEL
LIN {X 0,Y 340.714,Z 315.539,A -85,B 0,C 180,E1 -14264.532,E2 -14264.532} C_VEL
LIN {X 0,Y 340.692,Z 315.504,A -85,B 0,C 180,E1 -14268.692,E2 -14268.692} C_VEL
LIN {X 0,Y 340.731,Z 315.542,A -85,B 0,C 180,E1 -14271.773,E2 -14271.773} C_VEL
LIN {X 0,Y 340.717,Z 315.513,A -85,B 0,C 180,E1 -14275.596,E2 -14275.596} C_VEL
LIN {X 0,Y 340.692,Z 315.544,A -85,B 0,C 180,E1 -14278.956,E2 -14278.956} C_VEL
LIN {X 0,Y 340.771,Z 315.536,A -85,B 0,C 180,E1 -14282.475,E2 -14282.475} C_VEL
LIN {X 0,Y 340.751,Z 315.541,A -85,B 0,C 180,E1 -14285.639,E2 -14285.639} C_VEL
LIN {X 0,Y 340.748,Z 315.652,A -85,B 0,C 180,E1 -14287.813,E2 -14287.813} C_VEL
LIN {X 0,Y 340.931,Z 316.491,A -85,B 0,C 180,E1 -14288.112,E2 -14288.112} C_VEL
LIN {X 0,Y 342.359,Z 319.227,A -85,B 0,C 180,E1 -14288.51,E2 -14288.51} C_VEL
LIN {X 0,Y 344.492,Z 321.262,A -85,B 0,C 180,E1 -14288.96,E2 -14288.96} C_VEL
LIN {X 0,Y 346.592,Z 324.476,A -85,B 0,C 180,E1 -14289.487,E2 -14289.487} C_VEL
LIN {X 0,Y 348.969,Z 326.852,A -85,B 0,C 180,E1 -14290.042,E2 -14290.042} C_VEL
LIN {X 0,Y 351.719,Z 330.334,A -85,B 0,C 180,E1 -14290.721,E2 -14290.721} C_VEL
LIN {X 0,Y 353.899,Z 332.488,A -85,B 0,C 180,E1 -14291.28,E2 -14291.28} C_VEL
LIN {X 0,Y 356.94,Z 336.085,A -85,B 0,C 180,E1 -14292.074,E2 -14292.074} C_VEL
LIN {X 0,Y 359.469,Z 338.432,A -85,B 0,C 180,E1 -14292.776,E2 -14292.776} C_VEL
LIN {X 0,Y 362.801,Z 342.103,A -85,B 0,C 180,E1 -14293.735,E2 -14293.735} C_VEL
LIN {X 0,Y 365.83,Z 344.598,A -85,B 0,C 180,E1 -14294.642,E2 -14294.642} C_VEL
LIN {X 0,Y 369.17,Z 348.335,A -85,B 0,C 180,E1 -14295.766,E2 -14295.766} C_VEL
LIN {X 0,Y 372.802,Z 351.224,A -85,B 0,C 180,E1 -14297.036,E2 -14297.036} C_VEL
LIN {X 0,Y 376.097,Z 354.714,A -85,B 0,C 180,E1 -14298.351,E2 -14298.351} C_VEL
LIN {X 0,Y 379.345,Z 357.079,A -85,B 0,C 180,E1 -14299.761,E2 -14299.761} C_VEL
LIN {X 0,Y 381.144,Z 358.142,A -85,B 0,C 180,E1 -14300.617,E2 -14300.617} C_VEL
LIN {X 0,Y 383.823,Z 361.326,A -85,B 0,C 180,E1 -14302.189,E2 -14302.189} C_VEL
LIN {X 0,Y 386.503,Z 363.377,A -85,B 0,C 180,E1 -14304.061,E2 -14304.061} C_VEL
LIN {X 0,Y 388.386,Z 364.414,A -85,B 0,C 180,E1 -14305.849,E2 -14305.849} C_VEL
LIN {X 0,Y 389.529,Z 364.798,A -85,B 0,C 180,E1 -14307.434,E2 -14307.434} C_VEL
LIN {X 0,Y 390.099,Z 365.222,A -85,B 0,C 180,E1 -14308.968,E2 -14308.968} C_VEL
LIN {X 0,Y 390.27,Z 365.151,A -85,B 0,C 180,E1 -14310,E2 -14310} C_VEL
LIN {X 0,Y 389.992,Z 365.113,A -85,B 0,C 180,E1 -14311.549,E2 -14311.549} C_VEL
LIN {X 0,Y 389.238,Z 364.656,A -85,B 0,C 180,E1 -14313.105,E2 -14313.105} C_VEL
LIN {X 0,Y 387.614,Z 364.061,A -85,B 0,C 180,E1 -14314.941,E2 -14314.941} C_VEL
LIN {X 0,Y 385.473,Z 362.706,A -85,B 0,C 180,E1 -14316.684,E2 -14316.684} C_VEL
LIN {X 0,Y 383.225,Z 360.719,A -85,B 0,C 180,E1 -14318.163,E2 -14318.163} C_VEL
